			(* Case 20 - PROGRAMMA[106] ASSE Z -> TRASLAZIONE A QUOTA DI FUORI INGOMBRO *)	
			20:	
				IF StepInto THEN
					Programma_Z[Z_PosFuoriIngombroVuotoLastra].Stato 			:= DA_ESEGUIRE;
					Programma_Z[Z_PosFuoriIngombroVuotoLastra].InterpolaAsse 	:= NO_INTERPOLAZIONE_ASSE;
					ProgrammaToModule_Z 										:= Programma_Z[Z_PosFuoriIngombroVuotoLastra];
					Ciclo^.Passo := 21;
					STEPDone := FALSE;
				END_IF
				
			(* Case 21 - Attesa completamento del comando MOVETOPOS o del raggiungimento quota di Pre-Movimento se abilitata la funzione*)
			21: 
				IF Programma_Z[Z_PosFuoriIngombroVuotoLastra].Stato = TERMINATO OR
					Asse_Z_InFinestraDiPassMode OR 
					QuotaAnticipoDinamicaZ_Raggiunta THEN
					Ciclo^.Passo := 22;
					STEPDone := TRUE;
				ELSIF Programma_Z[Z_PosFuoriIngombroVuotoLastra].Stato = INTERROTTO THEN
					Ciclo^.Passo := 21;										
				END_IF
				
			(* Case 22 - Vado a quota di fuori ingombro con X *)
			22: IF Programma_Z[Z_PosFuoriIngombroVuotoLastra].Stato = INTERROTTO THEN
					Ciclo^.Passo := 22;
				ELSE
					IF StepInto THEN	
						IF FuoriIngombroXNecessario THEN
							Programma_X[X_PosFuoriIngombroVuotoLastra].Stato 			:= DA_ESEGUIRE;
							Programma_X[X_PosFuoriIngombroVuotoLastra].InterpolaAsse 	:= NO_INTERPOLAZIONE_ASSE;
							ProgrammaToModule_X 										:= Programma_X[X_PosFuoriIngombroVuotoLastra];
							Ciclo^.Passo := 23;
						ELSE
							Ciclo^.Passo := 24;
						END_IF
						STEPDone := FALSE;
					END_IF									
				END_IF

			(* Case 23 - Attendo x fuori ingombro *)
			23:
				IF Programma_Z[Z_PosFuoriIngombroVuotoLastra].Stato = INTERROTTO OR
					Programma_X[X_PosFuoriIngombroVuotoLastra].Stato = INTERROTTO THEN
						Ciclo^.Passo := 23;
				ELSIF (Programma_X[X_PosFuoriIngombroVuotoLastra].Stato = TERMINATO OR 
					Asse_X_InFinestraDiPassMode) THEN	
						Ciclo^.Passo := 24;
						STEPDone := TRUE;									
				END_IF
		
				
			(* Case 24 - Vado a quota di fuori ingombro y e j  *)
			24:
				IF Programma_Z[Z_PosFuoriIngombroVuotoLastra].Stato = INTERROTTO OR 
					Programma_X[X_PosFuoriIngombroVuotoLastra].Stato = INTERROTTO THEN
						Ciclo^.Passo := 24;										
				ELSE
					IF StepInto THEN
						Programma_Y[Y_PosFuoriIngombroVuotoLastra].Stato 			:= DA_ESEGUIRE;
						Programma_Y[Y_PosFuoriIngombroVuotoLastra].InterpolaAsse 	:= INTERPOLAZIONE_ASSE;
						ProgrammaToModule_Y 										:= Programma_Y[Y_PosFuoriIngombroVuotoLastra];

						Programma_J[J_PosStartApproccioPrelLastra].Stato 			:= DA_ESEGUIRE;
						//Programma_J[J_PosStartApproccioPrelLastra].InterpolaAsse 	:= INTERPOLAZIONE_ASSE;
						Programma_J[J_PosStartApproccioPrelLastra].InterpolaAsse 	:= No_INTERPOLAZIONE_ASSE;
						ProgrammaToModule_J 										:= Programma_J[J_PosStartApproccioPrelLastra];

						IF NOT FuoriIngombroYNecessario THEN
							Programma_X[X_PosStartLentaPrelievoLastra].Stato 			:= DA_ESEGUIRE;
							Programma_X[X_PosStartLentaPrelievoLastra].InterpolaAsse 	:= INTERPOLAZIONE_ASSE;
							ProgrammaToModule_X 										:= Programma_X[X_PosStartLentaPrelievoLastra];
							Ciclo^.Passo := 41;
						ELSE
							Ciclo^.Passo := 25;
						END_IF
						StartInterpolazioneAssi^ 	:= TRUE; //Abilito l'interpolazione degli assi
						STEPDone 					:= FALSE;
					END_IF
				END_IF
				
			(* Case 25 - *)
			25: IF Programma_Z[Z_PosFuoriIngombroVuotoLastra].Stato = INTERROTTO OR  
					(Programma_X[X_PosStartLentaPrelievoLastra].Stato = INTERROTTO and not FuoriIngombroYNecessario) OR
					Programma_Y[Y_PosFuoriIngombroVuotoLastra].Stato = INTERROTTO OR
					Programma_J[J_PosStartApproccioPrelLastra].Stato = INTERROTTO THEN
						Ciclo^.Passo := 25;
				ELSIF (Programma_Y[Y_PosFuoriIngombroVuotoLastra].Stato = TERMINATO OR 
					Asse_Y_InFinestraDiPassMode) AND 
					(Programma_J[J_PosStartApproccioPrelLastra].Stato = TERMINATO OR 
					Asse_J_InFinestraDiPassMode) THEN	
						Ciclo^.Passo := 40;
						STEPDone := TRUE;									
				END_IF
				
				
			(* Case 40 - PROGRAMMA[] ASSE  -> X TRASLAZIONE A QUOTA DI START LENTA PRELIEVO LASTRA *)	
			40:	
				IF Programma_Z[Z_PosFuoriIngombroVuotoLastra].Stato = INTERROTTO OR
					Programma_Y[Y_PosFuoriIngombroVuotoLastra].Stato = INTERROTTO OR
					Programma_J[J_PosStartApproccioPrelLastra].Stato = INTERROTTO THEN
						Ciclo^.Passo := 40;										
				ELSE
					IF StepInto THEN
						Programma_X[X_PosStartLentaPrelievoLastra].Stato 			:= DA_ESEGUIRE;
						Programma_X[X_PosStartLentaPrelievoLastra].InterpolaAsse 	:= NO_INTERPOLAZIONE_ASSE;
						ProgrammaToModule_X 										:= Programma_X[X_PosStartLentaPrelievoLastra];
												
						StartInterpolazioneAssi^ := FALSE; //Abilito l'interpolazione degli assi
						Ciclo^.Passo := 41;
						STEPDone := FALSE;
					END_IF
				END_IF
			
			(* Case 41 -   *)	
			41:	
				IF Programma_Z[Z_PosFuoriIngombroVuotoLastra].Stato = INTERROTTO OR
					Programma_Y[Y_PosFuoriIngombroVuotoLastra].Stato = INTERROTTO OR
					Programma_J[J_PosStartApproccioPrelLastra].Stato = INTERROTTO OR
					Programma_X[X_PosStartLentaPrelievoLastra].Stato = INTERROTTO THEN
						Ciclo^.Passo := 41;										
				ELSE
					STEPDone := TRUE;
					IF StepInto THEN
						Ciclo^.Passo := 42;
						STEPDone := FALSE;
					END_IF
				END_IF
				
			(* Case 42 -  Attesa completamento del comando MOVETOPOS o del raggiungimento quota di Pre-Movimento se abilitata la funzione *)
			42: 
				IF Programma_Z[Z_PosFuoriIngombroVuotoLastra].Stato = INTERROTTO OR
					Programma_Y[Y_PosFuoriIngombroVuotoLastra].Stato = INTERROTTO OR
					Programma_J[J_PosStartApproccioPrelLastra].Stato = INTERROTTO OR
					Programma_X[X_PosStartLentaPrelievoLastra].Stato = INTERROTTO THEN
						Ciclo^.Passo := 42;	
				ELSIF (Programma_X[X_PosStartLentaPrelievoLastra].Stato 	= TERMINATO OR Asse_X_InFinestraDiPassMode) AND
					(Programma_Y[Y_PosFuoriIngombroVuotoLastra].Stato		= TERMINATO OR Asse_Y_InFinestraDiPassMode) AND
					Programma_Z[Z_PosFuoriIngombroVuotoLastra].Stato 		= TERMINATO AND// OR Asse_Z_InFinestraDiPassMode AND
					(Programma_J[J_PosStartApproccioPrelLastra].Stato 		= TERMINATO OR Asse_J_InFinestraDiPassMode) THEN
						Ciclo^.Passo := 50;
						STEPDone := TRUE;							
				END_IF
							
			(* Case 50 - PROGRAMMA[101] ASSE Z -> TRASLAZIONE A QUOTA AMMESSA IN VELOCE DI PRELIEVO PACCO  *)
			50:
				IF StepInto THEN
					Programma_Z[Z_PosStartLentaPrelievoLastra].Stato 			:= DA_ESEGUIRE;
					Programma_Z[Z_PosStartLentaPrelievoLastra].InterpolaAsse 	:= NO_INTERPOLAZIONE_ASSE;
					ProgrammaToModule_Z 										:= Programma_Z[Z_PosStartLentaPrelievoLastra];
					Ciclo^.Passo := 51;
					STEPDone := FALSE;
				END_IF

			(* Case 51 -  Attesa completamento del comando MOVETOPOS o del raggiungimento quota di Pre-Movimento se abilitata la funzione *)
			51: 
				IF Programma_Z[Z_PosStartLentaPrelievoLastra].Stato = INTERROTTO OR
					Programma_Y[Y_PosFuoriIngombroVuotoLastra].Stato = INTERROTTO OR
					Programma_J[J_PosStartApproccioPrelLastra].Stato = INTERROTTO OR
					Programma_X[X_PosStartLentaPrelievoLastra].Stato = INTERROTTO THEN
						Ciclo^.Passo := 51;									
				ELSE
					IF Programma_X[X_PosStartLentaPrelievoLastra].Stato 	= TERMINATO AND
						Programma_Y[Y_PosFuoriIngombroVuotoLastra].Stato	= TERMINATO AND
						Programma_J[J_PosStartApproccioPrelLastra].Stato 	= TERMINATO AND
							(Programma_Z[Z_PosStartLentaPrelievoLastra].Stato = TERMINATO )THEN//OR Asse_Z_InFinestraDiPassMode) THEN
							Ciclo^.Passo := 90;
							STEPDone := TRUE;
					END_IF	
				END_IF
				
			52:
				IF Programma_Z[Z_PosStartLentaPrelievoLastra].Stato = INTERROTTO OR
					Programma_Y[Y_PosFuoriIngombroVuotoLastra].Stato = INTERROTTO OR
					Programma_J[J_PosStartApproccioPrelLastra].Stato = INTERROTTO OR
					Programma_X[X_PosStartLentaPrelievoLastra].Stato = INTERROTTO THEN
						Ciclo^.Passo := 52;									
				ELSE
					IF Programma_X[X_PosStartLentaPrelievoLastra].Stato 	= TERMINATO AND
						Programma_Y[Y_PosFuoriIngombroVuotoLastra].Stato	= TERMINATO AND
						Programma_J[J_PosStartApproccioPrelLastra].Stato 	= TERMINATO AND
							(Programma_Z[Z_PosStartLentaPrelievoLastra].Stato = TERMINATO )THEN
							IF StepInto THEN
								Programma_Z[Z_PosPrelievoInLentaLastra].Stato 			:= DA_ESEGUIRE;
								Programma_Z[Z_PosPrelievoInLentaLastra].InterpolaAsse 	:= NO_INTERPOLAZIONE_ASSE;
								ProgrammaToModule_Z 									:= Programma_Z[Z_PosPrelievoInLentaLastra];
								Ciclo^.Passo := 53;
								STEPDone := FALSE;
							END_IF
					END_IF	
				END_IF			
						
			53:
				IF Programma_Z[Z_PosPrelievoInLentaLastra].Stato = INTERROTTO OR
					Programma_Y[Y_PosFuoriIngombroVuotoLastra].Stato = INTERROTTO OR
					Programma_J[J_PosStartApproccioPrelLastra].Stato = INTERROTTO OR
					Programma_X[X_PosStartLentaPrelievoLastra].Stato = INTERROTTO THEN
						Ciclo^.Passo := 53;									
				ELSE
					IF Programma_X[X_PosStartLentaPrelievoLastra].Stato 	= TERMINATO AND
						Programma_Y[Y_PosFuoriIngombroVuotoLastra].Stato	= TERMINATO AND
						Programma_J[J_PosStartApproccioPrelLastra].Stato 	= TERMINATO AND
							(Programma_Z[Z_PosPrelievoInLentaLastra].Stato = TERMINATO )THEN
							Ciclo^.Passo := 90;
							STEPDone := TRUE;
					END_IF	
				END_IF

			(* Case 90 - PROGRAMMA[] ASSE Y -> TRASLAZIONE IN Y FINO ALLA QUOTA AMMESSA IN VELOCE E ATTIVAZIONE ASPIRAZIONE *)
			90:
				IF Programma_Z[Z_PosStartLentaPrelievoLastra].Stato = INTERROTTO OR
					Programma_Y[Y_PosFuoriIngombroVuotoLastra].Stato = INTERROTTO OR
					Programma_J[J_PosStartApproccioPrelLastra].Stato = INTERROTTO OR
					Programma_X[X_PosStartLentaPrelievoLastra].Stato = INTERROTTO THEN
						Ciclo^.Passo := 90; 									
				ELSE
					IF StepInto THEN
						Programma_Y[Y_PosStartLentaPrelievoLastra].Stato 			:= DA_ESEGUIRE;
						Programma_Y[Y_PosStartLentaPrelievoLastra].InterpolaAsse 	:= NO_INTERPOLAZIONE_ASSE;
						ProgrammaToModule_Y 										:= Programma_Y[Y_PosStartLentaPrelievoLastra];
						TFParametersArrayClear(ADR(ParametersArray));
						ParametersArray.Parameters[0] := BOOL_TO_STRING(NOT PrelievoPezzoOrizzontale);//SE TRUE: pezzo prelevato da cavallina, altrimenti prelievo orizzontale
						TFCommandSend(CmdPRELOAD,ParametersArray,ModulePinza^.Cmd);//LANCIO COMANDO ASPIRAZIONE PINZA
						Ciclo^.Passo := 91;
						STEPDone := FALSE;
					END_IF
				END_IF	
	
			(* Case 91 -  Attesa completamento dei comandi *)
			91: 
				IF Programma_Y[Y_PosStartLentaPrelievoLastra].Stato = INTERROTTO OR 
					TFStateCodeGet(ModulePinza^.State) = StateERROR THEN
						Ciclo^.Passo := 91; 										
				ELSE
					IF (Programma_Y[Y_PosStartLentaPrelievoLastra].Stato = TERMINATO OR Asse_Y_InFinestraDiPassMode) AND
						TFStateCodeGet(ModulePinza^.State) = StatePRELOAD_END THEN
							Ciclo^.Passo := 100;
							STEPDone := FALSE;
					END_IF	
				END_IF
				
			(* Case 100 - Lancio Tasteggio J *)
			100:
				IF StepInto THEN
					IF HMI_AbilitaTasteggioRotazionePinza THEN
						TFParametersArrayClear(ADR(ParametersArray));
						TFCommandSend(CmdTASTEGGIO,ParametersArray,ModuleAx_J^.Cmd);//LANCIO COMANDO per tateggio inclinazione pinza
					END_IF
					//!!!!!!!!!!!!!!!NB!!!!!!!!!!!	ModuleAx_J^.IN_Stop := TRUE; //Fermo Comando di tasteggio
					Ciclo^.Passo := 101;
					STEPDone := FALSE;
				END_IF

			(* Case 101 -  Attesa completamento del comando DI TASTEGGIO DELLA J*)
			101: 
				IF TFStateCodeGet(ModulePinza^.State) = StateError THEN
					Ciclo^.Passo := 101;																
				ELSE
					IF (TFStateCodeGet(ModuleAX_J^.State) >= StateTASTEGGIO_RUN + 10 AND TFStateCodeGet(ModuleAX_J^.State) <= StateTASTEGGIO_END) OR NOT HMI_AbilitaTasteggioRotazionePinza THEN		
						IF PrelievoPezzoOrizzontale THEN
							Ciclo^.Passo := 150;
						ELSE
							Ciclo^.Passo := 110;	
						END_IF

						STEPDone := TRUE;
					END_IF	
				END_IF
			
			(* Case 110 - Tasteggio in direzione Y *)
			110:
				IF Programma_Z[Z_PosStartLentaPrelievoLastra].Stato = INTERROTTO OR
					Programma_Y[Y_PosFuoriIngombroVuotoLastra].Stato = INTERROTTO OR
					Programma_J[J_PosStartApproccioPrelLastra].Stato = INTERROTTO OR
					Programma_X[X_PosStartLentaPrelievoLastra].Stato = INTERROTTO OR
					TFStateCodeGet(ModulePinza^.State) = StateError THEN
					Ciclo^.Passo := 110;																
				ELSE
					IF StepInto THEN
							
						Programma_Y[Y_PosPrelievoInLentaLastra].Stato 			:= DA_ESEGUIRE;
						Programma_Y[Y_PosPrelievoInLentaLastra].InterpolaAsse 	:= NO_INTERPOLAZIONE_ASSE;
						ProgrammaToModule_Y 									:= Programma_Y[Y_PosPrelievoInLentaLastra];
						StartInterpolazioneAssi^ := FALSE; 
						Ciclo^.Passo := 115;
						STEPDone := FALSE;
					END_IF
				END_IF	

			(* Case 115 -  Attesa completamento del comando di tasteggio IN Y *)
			115: 
				IF TFStateCodeGet(ModulePinza^.State) = StateError OR 
					Programma_Y[Y_PosPrelievoInLentaLastra].Stato = INTERROTTO	THEN
						Ciclo^.Passo := 115;																
				ELSE
					IF Programma_Y[Y_PosPrelievoInLentaLastra].Stato = TERMINATO THEN//Pezzo in presa
							Ciclo^.Passo := 116;//dichiaro il ciclo terminato
							ModuleAx_J^.IN_Stop := TRUE; //Fermo Comando di tasteggio
							STEPDone := TRUE;
					END_IF	
				END_IF

			(* Case 116 - DISTACCO LASTRA *)
			116: 
					IF StepInto THEN
						Programma_Z[Z_PosDistaccoLastraInLentaLastra].Stato 			:= DA_ESEGUIRE;
						Programma_Z[Z_PosDistaccoLastraInLentaLastra].InterpolaAsse 	:= INTERPOLAZIONE_ASSE;
						ProgrammaToModule_Z 											:= Programma_Z[Z_PosDistaccoLastraInLentaLastra];

						Programma_Y[Y_PosDistaccoLastraInLentaLastra].Stato 			:= DA_ESEGUIRE;
						Programma_Y[Y_PosDistaccoLastraInLentaLastra].InterpolaAsse 	:= INTERPOLAZIONE_ASSE;
						ProgrammaToModule_Y 											:= Programma_Y[Y_PosDistaccoLastraInLentaLastra];

						//TFParametersArrayClear(ADR(ParametersArray));
						//TFCommandSend(CmdCheckPresence,ParametersArray,ModulePinza^.Cmd);
					
						StartInterpolazioneAssi^ := TRUE; //Abilito l'interpolazione degli assi
						Ciclo^.Passo := 117;
						STEPDone := FALSE;
					END_IF	

			(* Case 117 -  Attesa completamento del comando *)
			117: 
				IF Programma_Z[Z_PosDistaccoLastraInLentaLastra].Stato = INTERROTTO OR
					Programma_Y[Y_PosDistaccoLastraInLentaLastra].Stato = INTERROTTO THEN
						Ciclo^.Passo := 117;																
				ELSE
					IF Programma_Z[Z_PosDistaccoLastraInLentaLastra].Stato = TERMINATO AND 
						Programma_Y[Y_PosDistaccoLastraInLentaLastra].Stato = TERMINATO THEN //AND 
						//TFStateCodeGet(ModulePinza^.State) = StateCHECKPRESENCE_END THEN
						TFParametersArrayClear(ADR(ParametersArray));
						TFCommandSend(CmdCheckPresence,ParametersArray,ModulePinza^.Cmd);
						Ciclo^.Passo := 118;//1000;//CICLO TERMINATO
					END_IF
				END_IF

			(* Case 118 -  Attesa completamento del comando *)
			118:
				IF TFStateCodeGet(ModulePinza^.State) = StateCHECKPRESENCE_END THEN
					IF	ModulePinza^.StatoPinza.ElementoPrelevato THEN
						IF StepInto THEN
							Ciclo^.Passo := 1000;//CICLO TERMINATO
							ModuleAx_J^.IN_Stop := TRUE; //Fermo Comando di tasteggio
							STEPDone := FALSE;
							SupportoVuoto := FALSE;
						END_IF
					ELSIF NOT ModulePinza^.StatoPinza.ElementoPrelevato THEN
						IF NumeroTentativiPresaAttuali >= NumeroTentativiPresa THEN
							SupportoVuoto := TRUE;
							IF StepInto THEN
								Ciclo^.Passo := 1000;//CICLO TERMINATO
								ModuleAx_J^.IN_Stop := TRUE; //Fermo Comando di tasteggio
								STEPDone := FALSE;
							END_IF
						ELSE
							SupportoVuoto := FALSE;
							Ciclo^.Passo := 50;//torno a fare prelievo     52??
							NumeroTentativiPresaAttuali := NumeroTentativiPresaAttuali+1;
						END_IF
					END_IF
				ELSIF TFStateCodeGet(ModulePinza^.State) = StateERROR THEN
					Ciclo^.Passo := 118;
				END_IF	
				
			(* Case 150 - Tasteggio in direzione Z *)
			150: 
				IF Programma_Z[Z_PosStartLentaPrelievoLastra].Stato = INTERROTTO OR
					Programma_Y[Y_PosPrelievoInLentaLastra].Stato = INTERROTTO OR
					Programma_J[J_PosStartApproccioPrelLastra].Stato = INTERROTTO OR
					Programma_X[X_PosStartLentaPrelievoLastra].Stato = INTERROTTO THEN
						Ciclo^.Passo := 150;									
				ELSE
					
					IF StepInto THEN
						Programma_Z[Z_PosPrelievoInLentaLastra].Stato 			:= DA_ESEGUIRE;
						Programma_Z[Z_PosPrelievoInLentaLastra].InterpolaAsse 	:= NO_INTERPOLAZIONE_ASSE;
						ProgrammaToModule_Z 									:= Programma_Z[Z_PosPrelievoInLentaLastra];
	
						Ciclo^.Passo := 155;
						STEPDone := FALSE;
					END_IF	
				END_IF
		
			(* Case 155 -  Attesa completamento del comando del tasteggio IN Z *)
			155: 
				IF TFStateCodeGet(ModulePinza^.State) = StateError OR 
					Programma_Z[Z_PosPrelievoInLentaLastra].Stato = INTERROTTO	THEN
						Ciclo^.Passo := 155;																
				ELSE
					IF Programma_Z[Z_PosPrelievoInLentaLastra].Stato = TERMINATO THEN//Pezzo in presa
						Ciclo^.Passo := 156;//VADO A ESEGUIRE IL DISTACCO LASTRA
						ModuleAx_J^.IN_Stop := TRUE; //Fermo Comando di tasteggio
						//TFParametersArrayClear(ADR(ParametersArray));
						//TFCommandSend(CmdCheckPresence,ParametersArray,ModulePinza^.Cmd);
						IF NumeroTentativiPresaAttuali = 0 THEN
							Programma_Z[Z_PosDistaccoLastraInLentaLastra].Quota_Destinazione := ModuleAX_Z^.QuotaAsseLetturaTasteggio + OffsetDistacco.Lastra.Z;
						ELSE
							Programma_Z[Z_PosDistaccoLastraInLentaLastra].Quota_Destinazione := ModuleAX_Z^.QuotaAsseLetturaTasteggio + OffsetDistacco.Lastra.Z+100;
						END_IF
						//
						
						RichiestaEspulsionePerPolistirolo := FALSE;
						IF ModuleAX_Z^.QuotaAsseLetturaTasteggio <= (WorkArea[Mission.PPick].Z + 1100) THEN
							idxTasteg := idxTasteg+1;
							IF idxTasteg > 10 THEN
								idxTasteg := 1;
								MemoriaQuoteTasteggio := MemoriaQuoteTasteggioVuoto;
							END_IF
							MemoriaQuoteTasteggio[idxTasteg] := ModuleAX_Z^.QuotaAsseLetturaTasteggio;
							IF (idxTasteg >= HMI_NumeroTentativiPolistiroloSuPallet)THEN
								FOR i := 1 TO HMI_NumeroTentativiPolistiroloSuPallet DO
									IF ModuleAX_Z^.QuotaAsseLetturaTasteggio <= MemoriaQuoteTasteggio[i]+2 THEN
										RichiestaEspulsionePerPolistirolo := TRUE;
										//Errore := ErrMalfunzionamentoSensoriPresenzaPinza;
										idxTasteg := 0;
										MemoriaQuoteTasteggio := MemoriaQuoteTasteggioVuoto;
									END_IF
								END_FOR
							END_IF
						ELSE
							idxTasteg := 0;
							MemoriaQuoteTasteggio := MemoriaQuoteTasteggioVuoto;
						END_IF
						
						STEPDone := TRUE;
					END_IF	
				END_IF

			(* Case 156 - Sfogliatura J *)
			156: 
					IF StepInto THEN
						Programma_Z[Z_PosDistaccoLastraInLentaLastra].Stato 			:= DA_ESEGUIRE;
						Programma_Z[Z_PosDistaccoLastraInLentaLastra].InterpolaAsse 	:= NO_INTERPOLAZIONE_ASSE;
						ProgrammaToModule_Z 											:= Programma_Z[Z_PosDistaccoLastraInLentaLastra];
						IF HMI_AbilitaSfogliaturaJ THEN
							Programma_J[J_PosSfogliatura].Stato 			:= DA_ESEGUIRE;
							Programma_J[J_PosSfogliatura].InterpolaAsse 	:= NO_INTERPOLAZIONE_ASSE;
							ProgrammaToModule_J 							:= Programma_J[J_PosSfogliatura];
						END_IF			
						TFTimerSet(ADR(TimerAttesaCadutaLastra),HMI_TempoAttesaPartenzaDopoPrelievo, TRUE);			
						Ciclo^.Passo := 157;
						STEPDone := FALSE;
					END_IF	
					
			157:
				IF Programma_Z[Z_PosDistaccoLastraInLentaLastra].Stato = INTERROTTO OR Programma_Z[J_PosSfogliatura].Stato = INTERROTTO	THEN
					Ciclo^.Passo := 157;																
				ELSE	
					IF Programma_Z[Z_PosDistaccoLastraInLentaLastra].Stato = TERMINATO AND TFTimerDone(ADR(TimerAttesaCadutaLastra)) THEN
						TFParametersArrayClear(ADR(ParametersArray));
						TFCommandSend(CmdCheckPresence,ParametersArray,ModulePinza^.Cmd);
						Ciclo^.Passo := 158;	
					END_IF
				END_IF	
					

			(* Case 158 -  Attesa completamento del comando *)
			158: 
				IF Programma_Z[Z_PosDistaccoLastraInLentaLastra].Stato = INTERROTTO OR Programma_Z[J_PosSfogliatura].Stato = INTERROTTO	THEN
						Ciclo^.Passo := 158;																
				ELSE
					//TFTimerSet(ADR(TimerAttesaCadutaLastra),HMI_TempoAttesaPartenzaDopoPrelievo, (Programma_Z[Z_PosDistaccoLastraInLentaLastra].Stato <> TERMINATO));
					IF Programma_Z[Z_PosDistaccoLastraInLentaLastra].Stato = TERMINATO AND TFTimerDone(ADR(TimerAttesaCadutaLastra)) AND
						TFStateCodeGet(ModulePinza^.State) = StateCHECKPRESENCE_END AND (Programma_J[J_PosSfogliatura].Stato = TERMINATO OR NOT HMI_AbilitaSfogliaturaJ) THEN
						IF ModulePinza^.StatoPinza.ElementoPrelevato AND NOT RichiestaEspulsionePerPolistirolo THEN
							Ciclo^.Passo := 1000;//CICLO TERMINATO
								
							ModuleAx_J^.IN_Stop := TRUE; //Fermo Comando di tasteggio
							STEPDone := FALSE;
							SupportoVuoto := FALSE;
							IF //((ModulePinza^.StatoPinza.LatoSxPiastrellaInPresa or ModulePinza^.StatoPinza.LatoDxPiastrellaInPresa) //AND 
								//(ModulePinza^.StatoPinza.LatoDxFaldaInPresa OR ModulePinza^.StatoPinza.LatoSxFaldaInPresa)) OR 
								(ModulePinza^.StatoPinza.LatoSxPiastrellaInPresa AND WorkAreaState[Mission.PPick].TransportState.Supporto.Tipologia = PALLET_STANDARD AND WorkAreaState[Mission.PPick].TransportState.Supporto.XDim < 1400 )OR
								(ModulePinza^.StatoPinza.LatoSxPiastrellaInPresa AND ModulePinza^.StatoPinza.LatoDxPiastrellaInPresa) THEN
									idxTasteg := 0;
									MemoriaQuoteTasteggio := MemoriaQuoteTasteggioVuoto;
							END_IF		
						ELSIF NOT ModulePinza^.StatoPinza.ElementoPrelevato OR (RichiestaEspulsionePerPolistirolo AND ModuleAX_Z^.QuotaAsseLetturaTasteggio <= (WorkArea[Mission.PPick].Z + HMI_AltezzaControlloPolistirolo)) THEN
							IF NumeroTentativiPresaAttuali >= NumeroTentativiPresa OR RichiestaEspulsionePerPolistirolo THEN
								idxTasteg := 0;
								MemoriaQuoteTasteggio := MemoriaQuoteTasteggioVuoto;
								SupportoVuoto := TRUE;
								RichiestaEspulsionePerPolistirolo := FALSE;
								IF StepInto THEN
									Ciclo^.Passo := 1000;//CICLO TERMINATO
									ModuleAx_J^.IN_Stop := TRUE; //Fermo Comando di tasteggio
									STEPDone := FALSE;
								END_IF
							ELSE
								SupportoVuoto := FALSE;
								Ciclo^.Passo := 150;//torno a fare prelievo
								NumeroTentativiPresaAttuali := NumeroTentativiPresaAttuali+1;
							END_IF
						ELSIF RichiestaEspulsionePerPolistirolo THEN
							idxTasteg := 0;
							MemoriaQuoteTasteggio := MemoriaQuoteTasteggioVuoto;
							RichiestaEspulsionePerPolistirolo := FALSE;
							Errore := ErrMalfunzionamentoSensoriPresenzaPinza;
						END_IF	
					END_IF
				END_IF	

			(* Case 159 - SFOGLIO J *)
			159: 
				IF StepInto THEN
					
					Programma_J[J_PosSfogliatura].Stato 			:= DA_ESEGUIRE;
					Programma_J[J_PosSfogliatura].InterpolaAsse 	:= NO_INTERPOLAZIONE_ASSE;
					ProgrammaToModule_J 							:= Programma_J[J_PosSfogliatura];
	
					Ciclo^.Passo := 159;
					STEPDone := FALSE;
				END_IF	

			(* Case 160 - FINE SFOGLIO J *)
			160:
				IF Programma_Z[J_PosSfogliatura].Stato = INTERROTTO	THEN
						Ciclo^.Passo := 160;																
				ELSE
					IF Programma_Z[J_PosSfogliatura].Stato = TERMINATO THEN//Pezzo in presa
						Ciclo^.Passo 		:= 1000;//termino ciclo
						ModuleAx_J^.IN_Stop := TRUE; //Fermo Comando di tasteggio
						STEPDone := TRUE;
					END_IF	
				END_IF

			(* Case 1000 *)
			1000:
				STEPDone := TRUE;
				Ciclo^.Stato := TERMINATO;
				Ciclo^.Passo := 1000;
				
			(* Case 9999 - Ciclo NON annullato o NON terminato*)
			9999:
				Ciclo^.Stato := INTERROTTO;
				Ciclo^.Passo := 9999;
	ELSE						
		;	
	END_CASE;
ELSE								//Se il ciclo deve essere interrotto, setto il suo nuovo stato
	Ciclo^.Stato := INTERROTTO;
END_IF

END_FUNCTION_BLOCK

// ---- POUs/TFCicliDiLavoro/Lastre/Cicli Depallettizzatore/TFCiclo_Deposito_Lastra_Depal.TcPOU
FUNCTION_BLOCK TFCiclo_Deposito_Lastra_Depal
VAR_INPUT
	Ciclo 		: POINTER TO Stato_Ciclo_Lavoro;
	Programma : POINTER TO TFProgramma_Ciclo_Lastra;
	ModuleAX_X : POINTER TO TFModulePalletizer_Ax;
	ModuleAX_Y : POINTER TO TFModulePalletizer_Ax;
	ModuleAX_Z : POINTER TO TFModulePalletizer_Ax;
	ModuleAX_J : POINTER TO TFModulePalletizer_AxJ_Lastre;
	ModulePinza : POINTER TO TFModulePalletizer_Pinza;
	StartInterpolazioneAssi : POINTER TO BOOL;
	QuotaPassModePuntoIntermedio : ARRAY [1..3] OF REAL;
	AbilitazioneGlobalePassMode	: BOOL;
	InterrompiCiclo : BOOL;
	Abilita_Ciclo_Step : BOOL;
	Command_Step : BOOL;
	AbilitazioneAnticipoDinamicoMovimenti : BOOL;
	
END_VAR
VAR_OUTPUT
	STEPDone	: BOOL;
	//MaterialeDepositatoSuLinea : BOOL;
END_VAR
VAR
	ConAccostamentoZ : BOOL := FALSE;
	StepInto: BOOL;
END_VAR

(* Set della variabile che mi permette di fare lo STEP nel ciclo *)
StepInto := (Abilita_Ciclo_Step AND Command_Step) OR NOT Abilita_Ciclo_Step;

(* Reset Anticipo Dinamico se non ho l'abilitazione *)
IF NOT AbilitazioneAnticipoDinamicoMovimenti OR NOT HMI_DisabilitaAnticipiGLOBALE THEN
	QuotaAnticipoDinamicaX_Raggiunta := FALSE;
	QuotaAnticipoDinamicaY_Raggiunta := FALSE;
	QuotaAnticipoDinamicaZ_Raggiunta := FALSE;
END_IF

IF NOT InterrompiCiclo THEN
	IF Ciclo^.Stato = TERMINATO OR Ciclo^.Stato = ANNULLATO THEN
		Ciclo^.Passo := 0;
	ELSIF Ciclo^.Stato = INTERROTTO AND Ciclo^.Passo = 56 THEN
		Ciclo^.Passo := 56;
	ELSIF Ciclo^.Stato = INTERROTTO AND NOT Ciclo^.Passo = 56 THEN
		Ciclo^.Passo := 999;
	END_IF
	Ciclo^.Stato := IN_ESECUZIONE;
	CASE Ciclo^.Passo OF
			(* Case 0 *)
			0:  Ciclo^.Stato := IN_ESECUZIONE;
				Ciclo^.Passo := 10;
				STEPDone := FALSE;
				
			(* Case 10 -  *)
			10:	MaterialeDepositatoSuLinea := FALSE;
				Ciclo^.Passo := 20;
				
						
			(* Case 20 - PROGRAMMA[Z_PosFuoriIngombroCaricoLastra] ASSE Z -> TRASLAZIONE A QUOTA DI FUORI INGOMBRO CON lLASTRA A BORDO *)	
			20:	Ciclo^.Stato := IN_ESECUZIONE;
				IF StepInto THEN
					Programma_Z[Z_PosFuoriIngombroCaricoLastra].Stato 			:= DA_ESEGUIRE;
					Programma_Z[Z_PosFuoriIngombroCaricoLastra].InterpolaAsse 	:= NO_INTERPOLAZIONE_ASSE;
					ProgrammaToModule_Z 										:= Programma_Z[Z_PosFuoriIngombroCaricoLastra];
					Ciclo^.Passo := 21;
					STEPDone := FALSE;
				END_IF
				
			(* Case 21 - Attesa completamento del comando MOVETOPOS o del raggiungimento quota di Pre-Movimento se abilitata la funzione*)
			21: 
				IF Programma_Z[Z_PosFuoriIngombroCaricoLastra].Stato = INTERROTTO THEN
					Ciclo^.Passo := 21;		
				ELSIF Programma_Z[Z_PosFuoriIngombroCaricoLastra].Stato = TERMINATO OR
					Asse_Z_InFinestraDiPassMode THEN
					Ciclo^.Passo := 22; //Eseguo prima il Fuori Ingombro colonne con la J poi il resto dei posizionamenti
					STEPDone := TRUE;							
				END_IF
				
			22: IF Programma_Z[Z_PosFuoriIngombroCaricoLastra].Stato = INTERROTTO THEN
					 Ciclo^.Passo := 22;
				ELSIF Programma_Z[Z_PosFuoriIngombroCaricoLastra].Stato = TERMINATO OR 
						Asse_Z_InFinestraDiPassMode OR 
						QuotaAnticipoDinamicaZ_Raggiunta THEN
							IF StepInto THEN
								Programma_J[J_PosFuoriIngombro].Stato 			:= DA_ESEGUIRE;
								Programma_J[J_PosFuoriIngombro].InterpolaAsse 	:= NO_INTERPOLAZIONE_ASSE;
								ProgrammaToModule_J		 						:= Programma_J[J_PosFuoriIngombro];
								Ciclo^.Passo := 23;
								STEPDone := FALSE;
							END_IF									
				END_IF
			
			23: IF Programma_Z[Z_PosFuoriIngombroCaricoLastra].Stato = INTERROTTO OR 
					Programma_J[J_PosFuoriIngombro].Stato = INTERROTTO THEN
					 Ciclo^.Passo := 23;
				ELSIF (Programma_Z[Z_PosFuoriIngombroCaricoLastra].Stato = TERMINATO OR Asse_Z_InFinestraDiPassMode (*OR QuotaAnticipoDinamicaZ_Raggiunta*)) AND 
					(Programma_J[J_PosFuoriIngombro].Stato = TERMINATO OR Asse_J_InFinestraDiPassMode OR QuotaAnticipoDinamicaJ_Raggiunta) THEN
						Ciclo^.Passo := 24;
						STEPDone := TRUE;										
				END_IF	
							
				
			(* Case 24 - Scelgo in quale direzione devo muovermi per primo a seconda della disposizione delle postazioni *)	
			24:	
				CASE ASSE_DISPOSIZIONE_POSTAZIONI OF
					
					LUNGO_X:
							Ciclo^.Passo := 25;
				
					LUNGO_Y:	
							IF FuoriIngombroXNecessario THEN
								IF FuoriIngombroYNecessario THEN
									Ciclo^.Passo := 25;
								ELSE
									Ciclo^.Passo := 50;
								END_IF
								
							ELSE
								Ciclo^.Passo := 52;
							END_IF
			
				END_CASE
				
			(* Case 25 - Vado a quota di fuori ingombro con Y *)
			25:	IF Programma_Z[Z_PosFuoriIngombroCaricoLastra].Stato = INTERROTTO OR
					Programma_J[J_PosFuoriIngombro].Stato = INTERROTTO THEN
						Ciclo^.Passo := 25;										
				ELSE
					IF StepInto THEN
						Programma_Y[Y_PosFuoriIngombroCaricoLastra].Stato 			:= DA_ESEGUIRE;
						Programma_Y[Y_PosFuoriIngombroCaricoLastra].InterpolaAsse 	:= NO_INTERPOLAZIONE_ASSE;
						ProgrammaToModule_Y 										:= Programma_Y[Y_PosFuoriIngombroCaricoLastra];
						Ciclo^.Passo := 26;
						STEPDone := FALSE;
					END_IF
				END_IF
					
			(* Case 26 - Check se a quota di fuori ingombro con Y *)		
			26:	IF Programma_Y[Y_PosFuoriIngombroCaricoLastra].Stato = INTERROTTO OR 
					Programma_Z[Z_PosFuoriIngombroCaricoLastra].Stato = INTERROTTO OR 
					Programma_J[J_PosFuoriIngombro].Stato = INTERROTTO THEN
						Ciclo^.Passo := 26;
				ELSE	
					IF Programma_Y[Y_PosFuoriIngombroCaricoLastra].Stato = TERMINATO OR 
						Asse_Y_InFinestraDiPassMode THEN
							Ciclo^.Passo := 30;
							STEPDone := TRUE;							
					END_IF
				END_IF
										
			(* Case 30 - PROGRAMMA[0] ASSE X  -> TRASLAZIONE A QUOTA DI DEPOSITO  *)	
			30:	IF Programma_Z[Z_PosFuoriIngombroCaricoLastra].Stato = INTERROTTO OR 
					Programma_Y[Y_PosFuoriIngombroCaricoLastra].Stato = INTERROTTO OR 
					Programma_J[J_PosFuoriIngombro].Stato = INTERROTTO THEN
						Ciclo^.Passo := 30;										
				ELSE
					IF StepInto THEN
						Programma_X[X_PosStartLentaDepositoLastra].Stato 			:= DA_ESEGUIRE;
						Programma_X[X_PosStartLentaDepositoLastra].InterpolaAsse 	:= NO_INTERPOLAZIONE_ASSE;
						ProgrammaToModule_X 										:= Programma_X[X_PosStartLentaDepositoLastra];
					
						Ciclo^.Passo := 31;
						STEPDone := FALSE;
					END_IF
				END_IF			
				
			(* Case 31 -  Attesa completamento del comando MOVETOPOS o del raggiungimento quota di Pre-Movimento se abilitata la funzione *)
			31: 
				IF Programma_X[X_PosStartLentaDepositoLastra].Stato = INTERROTTO OR
					Programma_Y[Y_PosFuoriIngombroCaricoLastra].Stato = INTERROTTO OR
					Programma_Z[Z_PosFuoriIngombroCaricoLastra].Stato = INTERROTTO OR 
					Programma_J[J_PosFuoriIngombro].Stato = INTERROTTO THEN
						Ciclo^.Passo := 31;
				ELSE	
					IF (Programma_X[X_PosStartLentaDepositoLastra].Stato = TERMINATO OR Asse_X_InFinestraDiPassMode OR QuotaAnticipoDinamicaX_Raggiunta) THEN 
						Ciclo^.Passo := 32;
						STEPDone := TRUE;							
					END_IF
				END_IF
				
			(* Case 32 - Vado a quota di START LENTA CON GLI ASSI con Y,Z,J *)
			32:
				IF Programma_X[X_PosStartLentaDepositoLastra].Stato = INTERROTTO OR
					Programma_Y[Y_PosFuoriIngombroCaricoLastra].Stato = INTERROTTO OR
					Programma_Z[Z_PosFuoriIngombroCaricoLastra].Stato = INTERROTTO OR 
					Programma_J[J_PosFuoriIngombro].Stato = INTERROTTO THEN
						Ciclo^.Passo := 32;										
				ELSE
					IF StepInto THEN
						TFParametersArrayClear(ADR(ParametersArray));
						Programma_Y[Y_PosStartLentaDepositoLastra].Stato 			:= DA_ESEGUIRE;
						Programma_Y[Y_PosStartLentaDepositoLastra].InterpolaAsse 	:= INTERPOLAZIONE_ASSE;
						ProgrammaToModule_Y 										:= Programma_Y[Y_PosStartLentaDepositoLastra];
				
						Programma_Z[Z_PosStartLentaDepositoLastra].Stato 			:= DA_ESEGUIRE;
						Programma_Z[Z_PosStartLentaDepositoLastra].InterpolaAsse 	:= INTERPOLAZIONE_ASSE;
						ProgrammaToModule_Z 										:= Programma_Z[Z_PosStartLentaDepositoLastra];
						
						Programma_J[J_PosDepositoLastra].Stato 						:= DA_ESEGUIRE;
						Programma_J[J_PosDepositoLastra].InterpolaAsse 				:= INTERPOLAZIONE_ASSE;
						ProgrammaToModule_J 										:= Programma_J[J_PosDepositoLastra];
						
						StartInterpolazioneAssi^ := TRUE; //Abilito l'interpolazione degli assi
												
						Ciclo^.Passo := 33;
						STEPDone := FALSE;
					END_IF
				END_IF
			
			(* Case 33 - Attendo completamento comando o assi in finsetra *)
			33:
				IF Programma_Y[Y_PosStartLentaDepositoLastra].Stato = TERMINATO (*OR Asse_Y_InFinestraDiPassMode)*) AND 
					Programma_J[J_PosDepositoLastra].Stato = TERMINATO (*OR Asse_J_InFinestraDiPassMode)*) AND
					Programma_X[X_PosStartLentaDepositoLastra].Stato = TERMINATO (*OR Asse_X_InFinestraDiPassMode)*) AND 
					Programma_Z[Z_PosStartLentaDepositoLastra].Stato = TERMINATO (*OR Asse_Z_InFinestraDiPassMode)*) THEN
						Ciclo^.Passo := 34;
						STEPDone := TRUE;
				ELSIF Programma_Y[Y_PosStartLentaDepositoLastra].Stato = INTERROTTO OR 
					Programma_J[J_PosDepositoLastra].Stato = INTERROTTO OR 
					Programma_X[X_PosStartLentaDepositoLastra].Stato = INTERROTTO OR
					Programma_Z[Z_PosStartLentaDepositoLastra].Stato = TERMINATO THEN

						Ciclo^.Passo := 33;								
				END_IF

			(* Case 34 - Vado a quota di finale con Z *)
			34:
				IF Programma_X[X_PosStartLentaDepositoLastra].Stato = INTERROTTO OR
					Programma_Y[Y_PosFuoriIngombroCaricoLastra].Stato = INTERROTTO OR
					Programma_Z[Z_PosFuoriIngombroCaricoLastra].Stato = INTERROTTO OR 
					Programma_J[J_PosFuoriIngombro].Stato = INTERROTTO THEN
						Ciclo^.Passo := 34;										
				ELSE
					IF StepInto THEN
						TFParametersArrayClear(ADR(ParametersArray));
						//Programma_Y[Y_PosDepositoInLentaLastra].Stato 			:= DA_ESEGUIRE;
						//Programma_Y[Y_PosDepositoInLentaLastra].InterpolaAsse 	:= INTERPOLAZIONE_ASSE;
						//ProgrammaToModule_Y 									:= Programma_Y[Y_PosDepositoInLentaLastra];
				
						Programma_Z[Z_PosDepositoInLentaLastra].Stato 			:= DA_ESEGUIRE;
						Programma_Z[Z_PosDepositoInLentaLastra].InterpolaAsse 	:= INTERPOLAZIONE_ASSE;
						ProgrammaToModule_Z 									:= Programma_Z[Z_PosDepositoInLentaLastra];
												
						StartInterpolazioneAssi^ := TRUE; //Abilito l'interpolazione degli assi
												
						Ciclo^.Passo := 35;
						STEPDone := FALSE;
					END_IF
				END_IF

			(* Case 35 - Attendo completamento comando o assi in finsetra *)
			35:
				IF //Programma_Y[Y_PosStartLentaDepositoLastra].Stato = TERMINATO (*OR Asse_Y_InFinestraDiPassMode)*) AND 
					//Programma_J[J_PosDepositoLastra].Stato = TERMINATO (*OR Asse_J_InFinestraDiPassMode)*) AND
					//Programma_X[X_PosStartLentaDepositoLastra].Stato = TERMINATO (*OR Asse_X_InFinestraDiPassMode)*) AND 
					Programma_Z[Z_PosDepositoInLentaLastra].Stato = TERMINATO (*OR Asse_Z_InFinestraDiPassMode)*) THEN
						Ciclo^.Passo := 90;
						STEPDone := TRUE;
				ELSIF //Programma_Y[Y_PosStartLentaDepositoLastra].Stato = INTERROTTO OR 
					//Programma_J[J_PosDepositoLastra].Stato = INTERROTTO OR 
					//Programma_X[X_PosStartLentaDepositoLastra].Stato = INTERROTTO OR
					Programma_Z[Z_PosDepositoInLentaLastra].Stato = INTERROTTO THEN
						Ciclo^.Passo := 35;								
				END_IF
										
			(* Case 50 - Vado a quota di deposito con X *)
			50:	IF Programma_Z[Z_PosFuoriIngombroCaricoLastra].Stato = INTERROTTO OR
					Programma_J[J_PosFuoriIngombro].Stato = INTERROTTO THEN
						Ciclo^.Passo := 50;										
				ELSE
					IF StepInto THEN
						Programma_X[X_PosStartLentaDepositoLastra].Stato 			:= DA_ESEGUIRE;
						Programma_X[X_PosStartLentaDepositoLastra].InterpolaAsse 	:= NO_INTERPOLAZIONE_ASSE;
						ProgrammaToModule_X 										:= Programma_X[X_PosStartLentaDepositoLastra];
						Ciclo^.Passo := 51;
						STEPDone := FALSE;
					END_IF
				END_IF
					
			(* Case 51 - Check se a quota di deposito X *)		
			51:	IF Programma_X[X_PosStartLentaDepositoLastra].Stato = INTERROTTO OR 
					Programma_Z[Z_PosFuoriIngombroCaricoLastra].Stato = INTERROTTO OR 
					Programma_J[J_PosFuoriIngombro].Stato = INTERROTTO THEN
						Ciclo^.Passo := 51;
				ELSE	
					IF Programma_X[X_PosStartLentaDepositoLastra].Stato = TERMINATO OR 
						Asse_X_InFinestraDiPassMode THEN
							Ciclo^.Passo := 52;
							STEPDone := TRUE;							
					END_IF
				END_IF
										
			(* Case 52 - lancio posizionamento Y,j e x se non serve fuori ingombro  *)	
			52:	IF Programma_Z[Z_PosFuoriIngombroCaricoLastra].Stato = INTERROTTO OR 
					(Programma_X[X_PosStartLentaDepositoLastra].Stato = INTERROTTO AND FuoriIngombroXNecessario) OR 
					Programma_J[J_PosFuoriIngombro].Stato = INTERROTTO THEN
						Ciclo^.Passo := 52;										
				ELSE
					IF StepInto THEN
			
						IF NOT FuoriIngombroXNecessario THEN
							Programma_X[X_PosStartLentaDepositoLastra].Stato 			:= DA_ESEGUIRE;
							Programma_X[X_PosStartLentaDepositoLastra].InterpolaAsse 	:= INTERPOLAZIONE_ASSE;
							ProgrammaToModule_X 										:= Programma_X[X_PosStartLentaDepositoLastra];
						END_IF
					
						Programma_Y[Y_PosStartLentaDepositoLastra].Stato 			:= DA_ESEGUIRE;
						Programma_Y[Y_PosStartLentaDepositoLastra].InterpolaAsse 	:= INTERPOLAZIONE_ASSE;
						ProgrammaToModule_Y 										:= Programma_Y[Y_PosStartLentaDepositoLastra];
						
						//Programma_Z[Z_PosStartLentaDepositoLastra].Stato 			:= DA_ESEGUIRE;
						//Programma_Z[Z_PosStartLentaDepositoLastra].InterpolaAsse 	:= INTERPOLAZIONE_ASSE;
						//ProgrammaToModule_Z 										:= Programma_Z[Z_PosStartLentaDepositoLastra];
					
					
						Programma_J[J_PosDepositoLastra].Stato 						:= DA_ESEGUIRE;
						Programma_J[J_PosDepositoLastra].InterpolaAsse 				:= INTERPOLAZIONE_ASSE;
						ProgrammaToModule_J 										:= Programma_J[J_PosDepositoLastra];
			
						StartInterpolazioneAssi^ := TRUE; //Abilito l'interpolazione degli assi

						Ciclo^.Passo := 53;
						STEPDone := FALSE;
					END_IF
				END_IF			
				
			(* Case 53 -  Attesa completamento del comando MOVETOPOS o del raggiungimento quota di Pre-Movimento se abilitata la funzione *)
			53: 
				IF Programma_X[X_PosStartLentaDepositoLastra].Stato = INTERROTTO OR
					Programma_Y[Y_PosStartLentaDepositoLastra].Stato = INTERROTTO OR
					Programma_Z[Z_PosFuoriIngombroCaricoLastra].Stato = INTERROTTO OR 
					Programma_J[J_PosDepositoLastra].Stato = INTERROTTO THEN
						Ciclo^.Passo := 53;
				ELSE	
					IF (Programma_Y[Y_PosStartLentaDepositoLastra].Stato = TERMINATO OR Asse_Y_InFinestraDiPassMode OR QuotaAnticipoDinamicaY_Raggiunta) AND
						(Programma_J[J_PosDepositoLastra].Stato = TERMINATO OR Asse_J_InFinestraDiPassMode OR QuotaAnticipoDinamicaJ_Raggiunta)  THEN 
							
							Ciclo^.Passo := 54;
							STEPDone := TRUE;							
					END_IF
				END_IF
				
			(* Case 54 - Vado a quota di START LENTA CON GLI ASSI Z*)
			54:
				IF Programma_X[X_PosStartLentaDepositoLastra].Stato = INTERROTTO OR
					Programma_Y[Y_PosStartLentaDepositoLastra].Stato = INTERROTTO OR
					//Programma_Z[Z_PosStartLentaDepositoLastra].Stato = INTERROTTO OR 
					Programma_J[J_PosDepositoLastra].Stato = INTERROTTO THEN
						Ciclo^.Passo := 54;										
				ELSE
					IF StepInto THEN
						Programma_Z[Z_PosStartLentaDepositoLastra].Stato 			:= DA_ESEGUIRE;
						Programma_Z[Z_PosStartLentaDepositoLastra].InterpolaAsse 	:= NO_INTERPOLAZIONE_ASSE;
						ProgrammaToModule_Z 										:= Programma_Z[Z_PosStartLentaDepositoLastra];
								
						Ciclo^.Passo := 55;
						STEPDone := FALSE;
					END_IF
				END_IF
			
			(* Case 55 - Attendo completamento comando o assi in finsetra *)
			55:
				IF Programma_Y[Y_PosStartLentaDepositoLastra].Stato = TERMINATO (*OR Asse_Y_InFinestraDiPassMode)*) AND 
					Programma_J[J_PosDepositoLastra].Stato = TERMINATO (*OR Asse_J_InFinestraDiPassMode)*) AND
					Programma_X[X_PosStartLentaDepositoLastra].Stato = TERMINATO (*OR Asse_X_InFinestraDiPassMode)*) AND 
					Programma_Z[Z_PosStartLentaDepositoLastra].Stato = TERMINATO OR Asse_Z_InFinestraDiPassMode THEN
						Ciclo^.Passo := 56;
						StopDepositoPerArresto := TRUE;
						STEPDone := TRUE;
				ELSIF Programma_X[X_PosStartLentaDepositoLastra].Stato = INTERROTTO OR
					Programma_Y[Y_PosStartLentaDepositoLastra].Stato = INTERROTTO OR
					Programma_Z[Z_PosFuoriIngombroCaricoLastra].Stato = INTERROTTO OR 
					Programma_J[J_PosDepositoLastra].Stato = INTERROTTO THEN
						Ciclo^.Passo := 55;
				END_IF

			(* Case 56 - Vado a quota di finale con Y,Z,J *)
			56:
				IF Programma_X[X_PosStartLentaDepositoLastra].Stato = INTERROTTO OR
					Programma_Y[Y_PosFuoriIngombroCaricoLastra].Stato = INTERROTTO OR
					Programma_Z[Z_PosFuoriIngombroCaricoLastra].Stato = INTERROTTO OR 
					Programma_J[J_PosFuoriIngombro].Stato = INTERROTTO THEN
						Ciclo^.Passo := 56;										
				ELSE
					IF StepInto THEN
						TFParametersArrayClear(ADR(ParametersArray));
						RichiestaDepositoALinea := TRUE;
						StopDepositoPerArresto := TRUE;
						IF OkDepositoDaLinea THEN
							Programma_Z[Z_PosDepositoInLentaLastra].Stato 			:= DA_ESEGUIRE;
							Programma_Z[Z_PosDepositoInLentaLastra].InterpolaAsse 	:= NO_INTERPOLAZIONE_ASSE;
							ProgrammaToModule_Z 									:= Programma_Z[Z_PosDepositoInLentaLastra];						
							Ciclo^.Passo := 57;
							STEPDone := FALSE;
						END_IF						
						//StartInterpolazioneAssi^ := TRUE; //Abilito l'interpolazione degli assi
						
					END_IF
				END_IF

			(* Case 57 - Attendo completamento comando o assi in finsetra *)
			57:
				IF //Programma_Y[Y_PosStartLentaDepositoLastra].Stato = TERMINATO (*OR Asse_Y_InFinestraDiPassMode)*) AND 
					//Programma_J[J_PosDepositoLastra].Stato = TERMINATO (*OR Asse_J_InFinestraDiPassMode)*) AND
					//Programma_X[X_PosStartLentaDepositoLastra].Stato = TERMINATO (*OR Asse_X_InFinestraDiPassMode)*) AND 
					Programma_Z[Z_PosDepositoInLentaLastra].Stato = TERMINATO (*OR Asse_Z_InFinestraDiPassMode)*) THEN
						Ciclo^.Passo := 90;
						STEPDone := TRUE;
				ELSIF //Programma_Y[Y_PosStartLentaDepositoLastra].Stato = INTERROTTO OR 
					//Programma_J[J_PosDepositoLastra].Stato = INTERROTTO OR 
					//Programma_X[X_PosStartLentaDepositoLastra].Stato = INTERROTTO OR
					Programma_Z[Z_PosDepositoInLentaLastra].Stato = INTERROTTO THEN

					Ciclo^.Passo := 57;								
				END_IF
						
			(* Case 90 - Attesa completamento posizionamento di tutti gli assi *)
			90: 
				IF TFStateCodeGet(ModulePinza^.State) = StateError THEN
					Ciclo^.Passo := 90;																
				ELSE
					RichiestaDepositoALinea := TRUE;
					IF StepInto AND OkDepositoDaLinea THEN
						TFParametersArrayClear(ADR(ParametersArray));
						TFCommandSend(CmdUNLOAD,ParametersArray,ModulePinza^.Cmd);
						Ciclo^.Passo := 91;
						STEPDone := FALSE;
					END_IF							
				END_IF

			(* Case 91 - Attesa completamento rilascio pezzo *)	
			91:
				IF TFStateCodeGet(ModulePinza^.State) = StateError THEN
					Ciclo^.Passo := 91;																
				ELSE
					STEPDone := TRUE;
					IF TFStateCodeGet(ModulePinza^.State) = StateUNLOAD_END THEN//Pezzo rilasciato
						RichiestaDepositoALinea := FALSE;
						Ciclo^.Passo := 92;//dichiaro il ciclo terminato
					END_IF	
				END_IF

			(* Case 92 - Vado in Fuori Ingombro con Z *)
			92:
				IF StepInto then//AND OkDepositoDaLinea THEN
					Programma_Z[Z_PosPostScarico].Stato 			:= DA_ESEGUIRE;
					Programma_Z[Z_PosPostScarico].InterpolaAsse 	:= NO_INTERPOLAZIONE_ASSE;
					ProgrammaToModule_Z 							:= Programma_Z[Z_PosPostScarico];
					Ciclo^.Passo := 93;
					STEPDone := FALSE;
				END_IF

			(* Case 93 - Attesa completamento del comando MOVETOPOS o del raggiungimento quota di Pre-Movimento se abilitata la funzione*)
			93: 
				IF Programma_Z[Z_PosPostScarico].Stato = TERMINATO THEN //OR
				//	Asse_Z_InFinestraDiPassMode OR 
				//	QuotaAnticipoDinamicaZ_Raggiunta THEN
					MaterialeDepositatoSuLinea := TRUE;
					Ciclo^.Passo := 1000;
					STEPDone := TRUE;
				ELSIF Programma_Z[Z_PosPostScarico].Stato = INTERROTTO THEN
					Ciclo^.Passo := 93;										
				END_IF

			(* Case 1000 *)
			1000:
				RichiestaDepositoALinea := FALSE;
				StopDepositoPerArresto := FALSE;
				Ciclo^.Stato := TERMINATO;
				Ciclo^.Passo := 1000;
				
			(* Case 9999 - Ciclo NON annullato o NON terminato*)
			9999:
				Ciclo^.Stato := INTERROTTO;
				Ciclo^.Passo := 9999;
	ELSE						
		;
			
	END_CASE;
ELSE								//Se il ciclo deve essere interrotto, setto il suo nuovo stato
	Ciclo^.Stato := INTERROTTO;
END_IF

END_FUNCTION_BLOCK

// ---- POUs/TFCicliDiLavoro/Lastre/Cicli Depallettizzatore/TFCiclo_Deposito_Falda_Depal.TcPOU
FUNCTION_BLOCK TFCiclo_Deposito_Falda_Depal
VAR_INPUT
	Ciclo 		: POINTER TO Stato_Ciclo_Lavoro;
	Programma  : POINTER TO TFProgramma_Ciclo_Falda_Lastre;
	ModuleAX_X : POINTER TO TFModulePalletizer_Ax;
	ModuleAX_Y : POINTER TO TFModulePalletizer_Ax;
	ModuleAX_Z : POINTER TO TFModulePalletizer_Ax;
	ModuleAX_J : POINTER TO TFModulePalletizer_AxJ_Lastre;
	StartInterpolazioneAssi : POINTER TO BOOL;
	//QuotaPassModePuntoIntermedio : ARRAY [1..3] OF REAL;
	ModulePinza : POINTER TO TFModulePalletizer_Pinza;
	TipoDiDeposito : UINT;
	AbilitazioneGlobalePassMode	: BOOL;
	InterrompiCiclo : BOOL;
	Abilita_Ciclo_Step : BOOL;
	Command_Step : BOOL;
	AbilitazioneAnticipoDinamicoMovimenti : BOOL;
END_VAR
VAR_OUTPUT
	STEPDone	: BOOL;
END_VAR
VAR
	StepInto: BOOL;
END_VAR

(* Set della variabile che mi permette di fare lo STEP nel ciclo *)
StepInto := (Abilita_Ciclo_Step AND Command_Step) OR NOT Abilita_Ciclo_Step;

(* Reset Anticipo Dinamico se non ho l'abilitazione *)
IF NOT AbilitazioneAnticipoDinamicoMovimenti  OR NOT HMI_DisabilitaAnticipiGLOBALE THEN
	QuotaAnticipoDinamicaX_Raggiunta := FALSE;
	QuotaAnticipoDinamicaY_Raggiunta := FALSE;
	QuotaAnticipoDinamicaZ_Raggiunta := FALSE;
END_IF

IF NOT InterrompiCiclo THEN
	IF Ciclo^.Stato = TERMINATO OR Ciclo^.Stato = ANNULLATO THEN
		Ciclo^.Passo := 0;
	ELSIF Ciclo^.Stato = INTERROTTO THEN
		Ciclo^.Passo := 999;
	END_IF
	Ciclo^.Stato := IN_ESECUZIONE;
	CASE Ciclo^.Passo OF
	(* Case 0 *)
			0:  Ciclo^.Stato := IN_ESECUZIONE;
				Ciclo^.Passo := 10;
				STEPDone := FALSE;
		
			(* Case 10 - *)	
			10:	
				Ciclo^.Passo := 11;
				
			(* Case 11 - *)
			11: 
				Ciclo^.Passo := 20;
				
			(* Case 20 - PROGRAMMA[54] ASSE Z -> TRASLAZIONE A QUOTA DI FUORI INGOMBRO *)	
			20:	Ciclo^.Stato := IN_ESECUZIONE;
				IF StepInto THEN
					Programma_Z[Z_PosFuoriIngombroFalda].Stato := DA_ESEGUIRE;
					Programma_Z[Z_PosFuoriIngombroFalda].InterpolaAsse := NO_INTERPOLAZIONE_ASSE;//FALSE;//NO_INTERPOLAZIONE_ASSE
					ProgrammaToModule_Z := Programma_Z[Z_PosFuoriIngombroFalda];
					Ciclo^.Passo := 21;
					STEPDone := FALSE;
				END_IF
				
			(* Case 21 - Attesa completamento del comando MOVETOPOS o del raggiungimento quota di Pre-Movimento se abilitata la funzione *)
			21: 
				IF Programma_Z[Z_PosFuoriIngombroFalda].Stato = TERMINATO OR 
					Asse_Z_InFinestraDiPassMode OR 
					QuotaAnticipoDinamicaZ_Raggiunta THEN
						Ciclo^.Passo := 22;
						STEPDone := TRUE;
				ELSIF Programma_Z[Z_PosFuoriIngombroFalda].Stato = INTERROTTO THEN
					Ciclo^.Passo := 21;										
				END_IF
				
			(* Case 22 - *)
			22:
				Ciclo^.Passo := 23;
				STEPDone := FALSE;
					
			(* Case 23 - *)		
			23:
				Ciclo^.Passo := 24;
				
			(* Case 24 - Scelgo in quale direzione devo muovermi per primo a seconda della disposizione delle postazioni *)	
			24:	
				CASE ASSE_DISPOSIZIONE_POSTAZIONI OF
					
					LUNGO_X:
							Ciclo^.Passo := 25;
				
					LUNGO_Y:	
							IF FuoriIngombroXNecessario THEN
								IF FuoriIngombroYNecessario THEN
									Ciclo^.Passo := 25;
								ELSE
									Ciclo^.Passo := 50;
								END_IF		
							ELSE
								Ciclo^.Passo := 50;
							END_IF
			
				END_CASE
				
			(* Case 25 - Vado a quota di fuori ingombro con Y *)
			25:	IF Programma_Z[Z_PosFuoriIngombroFalda].Stato = INTERROTTO THEN
					Ciclo^.Passo := 25;										
				ELSE
					IF StepInto THEN
						Programma_Y[Y_PosFuoriIngombroVuotoFalda].Stato 			:= DA_ESEGUIRE;
						Programma_Y[Y_PosFuoriIngombroVuotoFalda].InterpolaAsse 	:= NO_INTERPOLAZIONE_ASSE;
						ProgrammaToModule_Y 										:= Programma_Y[Y_PosFuoriIngombroVuotoFalda];
						Ciclo^.Passo := 26;
						STEPDone := FALSE;
					END_IF
				END_IF
					
			(* Case 26 - Check se a quota di fuori ingombro con Y *)		
			26:	IF Programma_Y[Y_PosFuoriIngombroVuotoFalda].Stato = INTERROTTO OR 
					Programma_Z[Z_PosFuoriIngombroFalda].Stato = INTERROTTO THEN
						Ciclo^.Passo := 26;
				ELSE	
					IF Programma_Y[Y_PosFuoriIngombroVuotoFalda].Stato = TERMINATO OR 
						Asse_Y_InFinestraDiPassMode THEN
							Ciclo^.Passo := 30;
							STEPDone := TRUE;							
					END_IF
				END_IF
										
			(* Case 30 - PROGRAMMA[0] ASSE X  -> TRASLAZIONE A QUOTA DI DEPOSITO  *)	
			30:	IF Programma_Z[Z_PosFuoriIngombroFalda].Stato = INTERROTTO OR 
					Programma_Y[Y_PosFuoriIngombroVuotoFalda].Stato = INTERROTTO THEN
						Ciclo^.Passo := 30;										
				ELSE
					IF StepInto THEN
						Programma_X[X_PosDepositoFalda].Stato 			:= DA_ESEGUIRE;
						Programma_X[X_PosDepositoFalda].InterpolaAsse 	:= NO_INTERPOLAZIONE_ASSE;
						ProgrammaToModule_X 							:= Programma_X[X_PosDepositoFalda];
						Ciclo^.Passo := 31;
						STEPDone := FALSE;
					END_IF
				END_IF			
				
			(* Case 31 -  Attesa completamento del comando MOVETOPOS o del raggiungimento quota di Pre-Movimento se abilitata la funzione *)
			31: 
				IF Programma_X[X_PosDepositoFalda].Stato = INTERROTTO OR
					Programma_Y[Y_PosFuoriIngombroVuotoFalda].Stato = INTERROTTO OR
					Programma_Z[Z_PosFuoriIngombroFalda].Stato = INTERROTTO THEN
						Ciclo^.Passo := 31;
				ELSE	
					IF (Programma_X[X_PosDepositoFalda].Stato = TERMINATO OR Asse_X_InFinestraDiPassMode OR QuotaAnticipoDinamicaX_Raggiunta) THEN 
						Ciclo^.Passo := 32;
						STEPDone := TRUE;							
					END_IF
				END_IF
				
			(* Case 32 - Vado a quota di START LENTA CON GLI ASSI con Y,Z,J *)
			32:
				IF Programma_X[X_PosDepositoFalda].Stato = INTERROTTO OR
					Programma_Y[Y_PosFuoriIngombroVuotoFalda].Stato = INTERROTTO OR
					Programma_Z[Z_PosFuoriIngombroFalda].Stato = INTERROTTO THEN
						Ciclo^.Passo := 32;										
				ELSE
					IF StepInto THEN
						TFParametersArrayClear(ADR(ParametersArray));
						Programma_Y[Y_PosDepositoFalda].Stato 			:= DA_ESEGUIRE;
						Programma_Y[Y_PosDepositoFalda].InterpolaAsse 	:= INTERPOLAZIONE_ASSE;
						ProgrammaToModule_Y 							:= Programma_Y[Y_PosDepositoFalda];
				
						//Programma_Z[Z_PosStartLentaDepositoLastra].Stato 			:= DA_ESEGUIRE;
						//Programma_Z[Z_PosStartLentaDepositoLastra].InterpolaAsse 	:= INTERPOLAZIONE_ASSE;
						//ProgrammaToModule_Z 										:= Programma_Z[Z_PosStartLentaDepositoLastra];
						
						Programma_J[J_PosDepositoFalda].Stato 						:= DA_ESEGUIRE;
						Programma_J[J_PosDepositoFalda].InterpolaAsse 				:= INTERPOLAZIONE_ASSE;
						ProgrammaToModule_J 										:= Programma_J[J_PosDepositoFalda];
						
						StartInterpolazioneAssi^ := TRUE; //Abilito l'interpolazione degli assi
												
						Ciclo^.Passo := 33;
						STEPDone := FALSE;
					END_IF
				END_IF
			
			(* Case 33 - Attendo completamento comando o assi in finsetra *)
			33:
				IF (Programma_X[X_PosDepositoFalda].Stato = TERMINATO OR Asse_X_InFinestraDiPassMode OR QuotaAnticipoDinamicaX_Raggiunta) AND
					(Programma_Y[Y_PosDepositoFalda].Stato = TERMINATO OR Asse_Y_InFinestraDiPassMode OR QuotaAnticipoDinamicaY_Raggiunta) AND
					(Programma_J[J_PosDepositoFalda].Stato = TERMINATO OR Asse_J_InFinestraDiPassMode OR QuotaAnticipoDinamicaJ_Raggiunta) THEN
						Ciclo^.Passo := 34;
						STEPDone := TRUE;
				ELSIF Programma_X[X_PosDepositoFalda].Stato = INTERROTTO OR
						Programma_Y[Y_PosDepositoFalda].Stato = INTERROTTO OR 
						Programma_J[J_PosDepositoFalda].Stato = INTERROTTO THEN
							Ciclo^.Passo := 33;								
				END_IF

			(* Case 34 - Vado a quota di finale con Z *)
			34:
				IF Programma_X[X_PosDepositoFalda].Stato = INTERROTTO OR
					Programma_Y[Y_PosDepositoFalda].Stato = INTERROTTO OR
					Programma_J[J_PosDepositoFalda].Stato = INTERROTTO THEN
						Ciclo^.Passo := 34;										
				ELSE
					IF StepInto THEN
						TFParametersArrayClear(ADR(ParametersArray));
				
						Programma_Z[Z_PosStartLentaDepositoFalda].Stato 			:= DA_ESEGUIRE;
						Programma_Z[Z_PosStartLentaDepositoFalda].InterpolaAsse 	:= INTERPOLAZIONE_ASSE;
						ProgrammaToModule_Z 													:= Programma_Z[Z_PosStartLentaDepositoFalda];
												
						StartInterpolazioneAssi^ := TRUE; //Abilito l'interpolazione degli assi
												
						Ciclo^.Passo := 35;
						STEPDone := FALSE;
					END_IF
				END_IF

			(* Case 35 - Attendo completamento comando o assi in finsetra *)
			35:
				IF //Programma_Y[Y_PosStartLentaDepositoLastra].Stato = TERMINATO (*OR Asse_Y_InFinestraDiPassMode)*) AND 
					//Programma_J[J_PosDepositoLastra].Stato = TERMINATO (*OR Asse_J_InFinestraDiPassMode)*) AND
					//Programma_X[X_PosStartLentaDepositoLastra].Stato = TERMINATO (*OR Asse_X_InFinestraDiPassMode)*) AND 
					Programma_Z[Z_PosStartLentaDepositoFalda].Stato = TERMINATO (*OR Asse_Z_InFinestraDiPassMode)*) THEN
						Ciclo^.Passo := 90;
						STEPDone := TRUE;
				ELSIF //Programma_Y[Y_PosStartLentaDepositoLastra].Stato = INTERROTTO OR 
					//Programma_J[J_PosDepositoLastra].Stato = INTERROTTO OR 
					//Programma_X[X_PosStartLentaDepositoLastra].Stato = INTERROTTO OR
					Programma_Z[Z_PosStartLentaDepositoFalda].Stato = INTERROTTO THEN
						Ciclo^.Passo := 35;								
				END_IF
										
			(* Case 50 - Vado a quota di fuori ingombro con X *)
			50:	IF Programma_Z[Z_PosFuoriIngombroFalda].Stato = INTERROTTO THEN
						Ciclo^.Passo := 50;										
				ELSE
					IF StepInto THEN
						Programma_X[X_PosDepositoFalda].Stato 			:= DA_ESEGUIRE;
						Programma_X[X_PosDepositoFalda].InterpolaAsse 	:= NO_INTERPOLAZIONE_ASSE;
						ProgrammaToModule_X 										:= Programma_X[X_PosDepositoFalda];
						Ciclo^.Passo := 51;
						STEPDone := FALSE;
					END_IF
				END_IF
					
			(* Case 51 - Check se a quota di fuori ingombro con Y *)		
			51:	IF Programma_X[X_PosDepositoFalda].Stato = INTERROTTO OR 
					Programma_Z[Z_PosFuoriIngombroFalda].Stato = INTERROTTO THEN
						Ciclo^.Passo := 51;
				ELSE	
					IF Programma_X[X_PosDepositoFalda].Stato = TERMINATO OR 
						Asse_X_InFinestraDiPassMode THEN
							Ciclo^.Passo := 52;
							STEPDone := TRUE;							
					END_IF
				END_IF
										
			(* Case 52 - lancio posizionamento Y+J e X se non serve il fuori ingombro  *)	
			52:	IF Programma_Z[Z_PosFuoriIngombroFalda].Stato = INTERROTTO OR 
					(Programma_X[X_PosDepositoFalda].Stato = INTERROTTO AND FuoriIngombroXNecessario) THEN
						Ciclo^.Passo := 52;										
				ELSE
					IF StepInto THEN
			
					//	IF NOT FuoriIngombroXNecessario THEN
						//	Programma_X[X_PosDepositoSuPostazioneFalda].Stato 			:= DA_ESEGUIRE;
						//	Programma_X[X_PosDepositoSuPostazioneFalda].InterpolaAsse 	:= INTERPOLAZIONE_ASSE;
						//	ProgrammaToModule_X 										:= Programma_X[X_PosDepositoSuPostazioneFalda];
					//	END_IF
					
						Programma_Y[Y_PosDepositoFalda].Stato 			:= DA_ESEGUIRE;
						Programma_Y[Y_PosDepositoFalda].InterpolaAsse 	:= INTERPOLAZIONE_ASSE;
						ProgrammaToModule_Y 										:= Programma_Y[Y_PosDepositoFalda];
						
						//Programma_Z[Z_PosStartLentaDepositoLastra].Stato 			:= DA_ESEGUIRE;
						//Programma_Z[Z_PosStartLentaDepositoLastra].InterpolaAsse 	:= INTERPOLAZIONE_ASSE;
						//ProgrammaToModule_Z 										:= Programma_Z[Z_PosStartLentaDepositoLastra];
					
						Programma_J[J_PosDepositoFalda].Stato 						:= DA_ESEGUIRE;
						Programma_J[J_PosDepositoFalda].InterpolaAsse 				:= INTERPOLAZIONE_ASSE;
						ProgrammaToModule_J 										:= Programma_J[J_PosDepositoFalda];
			
						StartInterpolazioneAssi^ := TRUE; //Abilito l'interpolazione degli assi

						Ciclo^.Passo := 53;
						STEPDone := FALSE;
					END_IF
				END_IF			
				
			(* Case 53 -  Attesa completamento del comando MOVETOPOS o del raggiungimento quota di Pre-Movimento se abilitata la funzione *)
			53: 
				IF Programma_X[X_PosDepositoFalda].Stato = INTERROTTO OR
					Programma_Y[Y_PosDepositoFalda].Stato = INTERROTTO OR
					Programma_Z[Z_PosFuoriIngombroFalda].Stato = INTERROTTO OR 
					Programma_J[J_PosDepositoFalda].Stato = INTERROTTO THEN
						Ciclo^.Passo := 53;
				ELSE	
					IF (Programma_Y[Y_PosDepositoFalda].Stato = TERMINATO OR Asse_Y_InFinestraDiPassMode OR QuotaAnticipoDinamicaY_Raggiunta) AND
						(Programma_J[J_PosDepositoFalda].Stato = TERMINATO OR Asse_J_InFinestraDiPassMode OR QuotaAnticipoDinamicaJ_Raggiunta)  THEN 	
							Ciclo^.Passo := 54;
							STEPDone := TRUE;							
					END_IF
				END_IF
				
			(* Case 54 - Vado a quota di START LENTA CON GLI ASSI Z*)
			54:
				IF Programma_X[X_PosDepositoFalda].Stato 	= INTERROTTO OR
					Programma_Y[Y_PosDepositoFalda].Stato 	= INTERROTTO OR
					Programma_Z[Z_PosFuoriIngombroFalda].Stato 	= INTERROTTO OR 
					Programma_J[J_PosDepositoFalda].Stato 				= INTERROTTO THEN
						Ciclo^.Passo := 54;										
				ELSE
					IF StepInto THEN
						Programma_Z[Z_PosStartLentaDepositoFalda].Stato 			:= DA_ESEGUIRE;
						Programma_Z[Z_PosStartLentaDepositoFalda].InterpolaAsse 	:= NO_INTERPOLAZIONE_ASSE;
						ProgrammaToModule_Z 										:= Programma_Z[Z_PosStartLentaDepositoFalda];
								
						Ciclo^.Passo := 55;
						STEPDone := FALSE;
					END_IF
				END_IF
			
			(* Case 55 - Attendo completamento comando o assi in finsetra *)
			55:
				IF Programma_Y[Y_PosDepositoFalda].Stato = TERMINATO (*OR Asse_Y_InFinestraDiPassMode)*) AND 
					Programma_J[J_PosDepositoFalda].Stato = TERMINATO (*OR Asse_J_InFinestraDiPassMode)*) AND
					Programma_X[X_PosDepositoFalda].Stato = TERMINATO (*OR Asse_X_InFinestraDiPassMode)*) AND 
					Programma_Z[Z_PosStartLentaDepositoFalda].Stato = TERMINATO OR Asse_Z_InFinestraDiPassMode THEN
						Ciclo^.Passo := 56;
						STEPDone := TRUE;
				ELSIF Programma_X[X_PosDepositoFalda].Stato 	= INTERROTTO OR
					Programma_Y[Y_PosDepositoFalda].Stato 	= INTERROTTO OR
					Programma_Z[Z_PosStartLentaDepositoFalda].Stato 	= INTERROTTO OR 
					Programma_J[J_PosDepositoFalda].Stato 				= INTERROTTO THEN
						Ciclo^.Passo := 55;
				END_IF

			(* Case 56 - Vado a quota di finale con Y,Z,J *)
			56:
				IF Programma_X[X_PosStartLentaDepositoLastra].Stato = INTERROTTO OR
					Programma_Y[Y_PosFuoriIngombroCaricoLastra].Stato = INTERROTTO OR
					Programma_Z[Z_PosFuoriIngombroCaricoLastra].Stato = INTERROTTO OR 
					Programma_J[J_PosFuoriIngombro].Stato = INTERROTTO THEN
						Ciclo^.Passo := 56;										
				ELSE
					IF StepInto THEN
						TFParametersArrayClear(ADR(ParametersArray));
						Programma_Z[Z_PosStartLentaDepositoFalda].Stato 			:= DA_ESEGUIRE;
						Programma_Z[Z_PosStartLentaDepositoFalda].InterpolaAsse 	:= NO_INTERPOLAZIONE_ASSE;
						ProgrammaToModule_Z 										:= Programma_Z[Z_PosStartLentaDepositoFalda];						
						Ciclo^.Passo := 57;
						STEPDone := FALSE;
					END_IF
				END_IF

			(* Case 57 - Attendo completamento comando o assi in finsetra *)
			57:
				IF Programma_Z[Z_PosStartLentaDepositoFalda].Stato = TERMINATO (*OR Asse_Z_InFinestraDiPassMode)*) THEN
					Ciclo^.Passo := 90;
					STEPDone := TRUE;
				ELSIF Programma_Z[Z_PosStartLentaDepositoFalda].Stato = INTERROTTO THEN
					Ciclo^.Passo := 57;								
				END_IF
						
			(* Case 90 - Attesa completamento posizionamento di tutti gli assi *)
			90: 
				IF TFStateCodeGet(ModulePinza^.State) = StateError THEN
					Ciclo^.Passo := 90;																
				ELSE
					IF StepInto THEN
						TFParametersArrayClear(ADR(ParametersArray));
						TFCommandSend(CmdUNLOAD,ParametersArray,ModulePinza^.Cmd);
						Ciclo^.Passo := 91;
						STEPDone := FALSE;
					END_IF							
				END_IF

			(* Case 91 - Attesa completamento rilascio pezzo *)	
			91:
				IF TFStateCodeGet(ModulePinza^.State) = StateError THEN
					Ciclo^.Passo := 91;																
				ELSE
					STEPDone := TRUE;
					IF TFStateCodeGet(ModulePinza^.State) = StateUNLOAD_END THEN//Pezzo rilasciato
						Ciclo^.Passo := 1000;//dichiaro il ciclo terminato
					END_IF	
				END_IF

			(* Case 1000 *)
			1000:
				Ciclo^.Stato := TERMINATO;
				Ciclo^.Passo := 1000;
				
			(* Case 9999 - Ciclo NON annullato o NON terminato*)
			9999:
				Ciclo^.Stato := INTERROTTO;
				Ciclo^.Passo := 9999;
	ELSE						
		;
			
	END_CASE;
ELSE								//Se il ciclo deve essere interrotto, setto il suo nuovo stato
	Ciclo^.Stato := INTERROTTO;
END_IF

END_FUNCTION_BLOCK

// ---- POUs/TFPalletizerDataTF/Utility Varie/TFCalcoloTraiettoriaLastre.TcPOU
FUNCTION_BLOCK TFCalcoloTraiettoriaLastre
VAR_INPUT
	Traiettoria : POINTER TO TFTraiettoria;
	WorkSpace : POINTER TO TFMachinePalletizer_WorkSpace;
	WorkFootprint : POINTER TO ARRAY [1..MAXFOOTPRINT] OF TFMachinePalletizer_WorkFootprint;
	WorkPickPoint : POINTER TO ARRAY [1..MAXPICKPOINT] OF TFMachinePalletizer_WorkPickPointSlab;
	WorkPickPointState : POINTER TO ARRAY [1..MAXPICKPOINT] OF TFMachinePalletizer_WorkPickPoint_State;
	WorkPickPointDimension 		: POINTER TO ARRAY [1..MAXPICKPOINT] OF Work_PickPoint_Dimension;

	WorkArea : POINTER TO ARRAY [1..MAXAREA] OF TFMachinePalletizer_WorkArea;
	WorkAreaState : POINTER TO ARRAY [1..MAXAREA] OF TFMachinePalletizer_WorkAreaState;
	Pallet : POINTER TO ARRAY [1..MAXPALLET] OF TFMachinePalletizer_Pallet;
	Layer : POINTER TO ARRAY [1..MAXLAYER] OF TFMachinePalletizer_Layer;
	Forming : POINTER TO ARRAY [1..MAXFORMING] OF TFMachinePalletizer_FormingForSlab;
	//ZDim : REAL;
	
	Mission : POINTER TO TFMachinePalletizer_Mission;
	
	WorkAreaManager : POINTER TO TFWorkAreaManager;
	ModuleAX_X : POINTER TO TFModulePalletizer_Ax;
	ModuleAX_Y : POINTER TO TFModulePalletizer_Ax;
	ModuleAX_Z : POINTER TO TFModulePalletizer_Ax;
	ModuleAX_J : POINTER TO TFModulePalletizer_AxJ_Lastre;
	//ModuleAX_K : POINTER TO TFModulePalletizer_Ax;
	Eseguito : BOOL;
	
END_VAR
VAR
	f : UINT;
	wa : UINT;
	P : UINT;
	a : uint;
	
	WASX : UINT;
	WADX : UINT;
	WAPARTENZA : UINT;
	WADESTINAZIONE : UINT;

	AltezzaDiIngombroArea_CCENTRALE : LREAL; //Altezza ingombro dell'Area nel corridoio CENTRALE
	AltezzaDiIngombroArea_CESTERNO : LREAL; //Altezza ingombro dell'Area nel corridoio ESTERNO
	AltezzaDiIngombroArea_CINTERNO : LREAL; //Altezza ingombro dell'Area nel corridoio INTERNO
	
	AltezzaDiIngombroIngombri_CCENTRALE : LREAL; //Altezza ingombro dell'Area nel corridoio CENTRALE
	AltezzaDiIngombroIngombri_CESTERNO : LREAL; //Altezza ingombro dell'Area nel corridoio ESTERNO
	AltezzaDiIngombroIngombri_CINTERNO : LREAL; //Altezza ingombro dell'Area nel corridoio INTERNO
	

	
	
	AltezzaDiIngombroOstacoli : LREAL;
	AltezzaDiIngombroPuntiPrelievo : LREAL;
	AssegnaQuote : BOOL;
	OffsetSicurezzaConPacco : REAL;
	AltezzaPinzaDaTastatoreAFlangiaMotore : REAL; // Altezza della pinza dal tastatore al bordo superiore della flangia di supporto motore asse K
	AltezzaDaPavimentoAPiastraSupportoColonnaCentrale : REAL;
	LarghezzaPiastraSupportoColonnaCentrale : REAL;
	Quota_X_CentroColonnaCentrale : REAL;
	
	


	(*
	IngombroX_Pos 	: LREAL;//Ingombro della pinza nella Metà POSITIVA della pinza lungo X
	IngombroY_Pos 	: LREAL;//Ingombro della pinza nella Metà POSITIVA della pinza lungo Y
	IngombroZ_Pos 	: LREAL;//Ingombro della pinza nella Metà POSITIVA della pinza lungo Z
	
	IngombroX_Neg 	: LREAL;//Ingombro della pinza nella Metà NEGATIVA della pinza lungo X
	IngombroY_Neg 	: LREAL;//Ingombro della pinza nella Metà NEGATIVA della pinza lungo Y
	IngombroZ_Neg 	: LREAL;//Ingombro della pinza nella Metà NEGATIVA della pinza lungo Z

	IngombroY_Tot 	: LREAL;//Ingombro totale In direzione Y
	*)
	debug : bool;
	CalcolaQuote : BOOL;
	AbilitaValutazioneFISuSingolaWA 		: BOOL;
	NumeroWAValutazioneFISingolaPostazione 	: UINT;
	//TFCalcolaNumeroPostazioneDXSX : TFCalcolaNumeroPostazioneDXSX;
	

END_VAR

(*(* Calcolo gli ingombri della pinza nelle varie direzioni *)
TFCalcoliIngombroPinza(Mission := Mission,
					WorkAreaManager := WorkAreaManager,
					ModuleAX_J := ModuleAX_J,
					AngoloRotazioneDestinazionePinza:= Mission^.JPick,
					IngombroX_Pos := ADR(IngombroX_Pos),
					IngombroY_Pos := ADR(IngombroY_Pos),
					IngombroX_Neg := ADR(IngombroX_Neg),
					IngombroY_Neg := ADR(IngombroY_Neg),
					IngombroZ_Pos := ADR(IngombroZ_Pos),
					IngombroZ_Neg := ADR(IngombroZ_Neg),
					IngombroY_Tot := ADR(IngombroY_Tot),
					IngombroDestinazioneX_Pos := ADR(IngombroDestinazioneX_Pos),
					IngombroDestinazioneY_Pos := ADR(IngombroDestinazioneY_Pos),
					IngombroDestinazioneX_Neg := ADR(IngombroDestinazioneX_Neg),
					IngombroDestinazioneY_Neg := ADR(IngombroDestinazioneY_Neg),
					IngombroDestinazioneZ_Pos := ADR(IngombroDestinazioneZ_Pos),
					IngombroDestinazioneZ_Neg := ADR(IngombroDestinazioneZ_Neg),
					IngombroMaxX_Pos := ADR(IngombroMaxX_Pos),
					IngombroMaxY_Pos := ADR(IngombroMaxY_Pos),
					IngombroMaxX_Neg := ADR(IngombroMaxX_Neg),
					IngombroMaxY_Neg := ADR(IngombroMaxY_Neg),
					IngombroMaxZ_Pos := ADR(IngombroMaxZ_Pos),
					IngombroMaxZ_Neg := ADR(IngombroMaxZ_Neg));*)

CASE WorkAreaManager^.State OF
	WAMANAGER_NOP:
		CalcolaQuote := TRUE;
	
	WAMANAGER_CICLO_RIPOSO_INIT:
		CalcolaQuote := TRUE;

{Region "Ciclo Riposo"}		
	WAMANAGER_CICLO_RIPOSO_RUN:

		IF CalcolaQuote THEN
			CalcolaQuote := FALSE;
			(*QuotaFuoriIngombro_Z_AVUOTO_CCENTRALE 	:= 0;
			QuotaFuoriIngombro_Z_AVUOTO_CESTERNO 	:= 0;
			QuotaFuoriIngombro_Z_AVUOTO_CINTERNO 	:= 0;
			AltezzaDiIngombroPuntiPrelievo := 0;
			AltezzaDiIngombroIngombri_CCENTRALE := 0;
			(* Valuto gli ostacoli *)	
			FOR f:=1 TO MAXFOOTPRINT DO
				AltezzaDiIngombroIngombri_CCENTRALE := MAX(AltezzaDiIngombroIngombri_CCENTRALE,WorkFootPrint^[f].Z + WorkFootPrint^[f].ZDim + IngombroMaxZ_Neg);
			END_FOR

			(* Valuto I Pick-Point *)
			FOR P:=1 TO MAXPICKPOINT DO	
				AltezzaDiIngombroPuntiPrelievo := MAX(AltezzaDiIngombroPuntiPrelievo,WorkPickPointDimension^[P].Zdim,WorkPickPoint^[P].ZRaise,WorkPickPoint^[P].Z);
			END_FOR

			(* Valuto le wa *)			
			CASE ASSE_DISPOSIZIONE_POSTAZIONI OF
				
				LUNGO_X:
						CalcolaIngombroWALungoX_Pal();
				
				LUNGO_Y:
						CalcolaIngombroWALungoY_Pal();
			
			END_CASE

			QuotaFuoriIngombro_Z_AVUOTO_CCENTRALE := MAX(AltezzaDiIngombroArea_CCENTRALE,AltezzaDiIngombroIngombri_CCENTRALE,AltezzaDiIngombroPuntiPrelievo) + IngombroMaxZ_Neg;
			QuotaFuoriIngombro_Z_AVUOTO_CESTERNO := MAX(AltezzaDiIngombroArea_CESTERNO,AltezzaDiIngombroIngombri_CCENTRALE,AltezzaDiIngombroPuntiPrelievo) + IngombroMaxZ_Neg;
			QuotaFuoriIngombro_Z_AVUOTO_CINTERNO := MAX(AltezzaDiIngombroArea_CINTERNO,AltezzaDiIngombroIngombri_CCENTRALE,AltezzaDiIngombroPuntiPrelievo) +IngombroMaxZ_Neg;
			QuotaFuoriIngombro_Z_AVUOTO := MAX(QuotaFuoriIngombro_Z_AVUOTO_CCENTRALE,QuotaFuoriIngombro_Z_AVUOTO_CESTERNO,QuotaFuoriIngombro_Z_AVUOTO_CINTERNO)+OffsetSicurezza.Z.Avuoto;
			*)
			(* Valuto se gli assi sono in finestra di prelievo, in questo modo valuto nel ciclo se devo andare fuori ingombro oppure posso partire da dove sono *)
			AsseXInFinestraDiPrelievo := FALSE;
			IF (ModuleAx_X^.Ax^.AxRef^.NcToPlc.ActPos >= Mission^.XPick - 50) AND (ModuleAx_X^.Ax^.AxRef^.NcToPlc.ActPos <=  Mission^.XPick + 50) THEN
				AsseXInFinestraDiPrelievo := TRUE;
			END_IF
			AsseYInFinestraDiPrelievo := FALSE;
			IF (ModuleAx_Y^.Ax^.AxRef^.NcToPlc.ActPos  >=  Mission^.YPick - 50) AND (ModuleAx_Y^.Ax^.AxRef^.NcToPlc.SetPos <= Mission^.YPick + 50) THEN
				AsseYInFinestraDiPrelievo := TRUE;
			END_IF
			(* Valuto la rotazione della pinza *)
			AsseJInFinestraDiPrelievo := FALSE;
			IF ModuleAx_J^.Ax^.AxRef^.NcToPlc.ActPos >= Mission^.JPick - 5 AND ModuleAx_J^.Ax^.AxRef^.NcToPlc.ActPos <= Mission^.JPick + 5 THEN
				AsseJInFinestraDiPrelievo := TRUE;
			END_IF
			
		END_IF

		//QuotaFuoriIngombro_Z_AVUOTO := MAX(QuotaFuoriIngombro_Z_AVUOTO_CCENTRALE,QuotaFuoriIngombro_Z_AVUOTO_CESTERNO,QuotaFuoriIngombro_Z_AVUOTO_CINTERNO)+OffsetSicurezza.Z.Avuoto;
		//QuotaFuoriIngombro_Z_ConPEZZO := MAX(QuotaFuoriIngombro_Z_AVUOTO_CCENTRALE,QuotaFuoriIngombro_Z_AVUOTO_CESTERNO,QuotaFuoriIngombro_Z_AVUOTO_CINTERNO)+OffsetSicurezza.Z.Carico;


	WAMANAGER_CICLO_RIPOSO_END:
		CalcolaQuote := TRUE;
{Endregion}

{Region "CCLO LASTRA PP"}
	WAMANAGER_CICLO_LASTRA_PP_INIT:
		CalcolaQuote := TRUE;

	WAMANAGER_CICLO_PRELIEVO_LASTRA_PP_RUN:
		
		IF CalcolaQuote THEN
			(*CalcolaQuote := FALSE;
			QuotaFuoriIngombro_Z_AVUOTO_CCENTRALE 	:= 0;
			QuotaFuoriIngombro_Z_AVUOTO_CESTERNO 	:= 0;
			QuotaFuoriIngombro_Z_AVUOTO_CINTERNO 	:= 0;
			AltezzaDiIngombroPuntiPrelievo := 0;
			AltezzaDiIngombroIngombri_CCENTRALE := 0;
			(* Valuto gli ostacoli *)	
			FOR f:=1 TO MAXFOOTPRINT DO
				AltezzaDiIngombroIngombri_CCENTRALE := MAX(AltezzaDiIngombroIngombri_CCENTRALE,WorkFootPrint^[f].Z + WorkFootPrint^[f].ZDim + IngombroMaxZ_Neg);
			END_FOR

			(* Valuto I Pick-Point *)
			FOR P:=1 TO MAXPICKPOINT DO	
				AltezzaDiIngombroPuntiPrelievo := MAX(AltezzaDiIngombroPuntiPrelievo,WorkPickPointDimension^[P].Zdim,WorkPickPoint^[P].ZRaise,WorkPickPoint^[P].Z);
			END_FOR
			//Per la postazione 2 valuto il FI solo della postazione stessa perchè non è in interferenza con la postazione n°1
			AbilitaValutazioneFISuSingolaWA 		:= FALSE;
			NumeroWAValutazioneFISingolaPostazione 	:= 0;
			//IF Mission^.PPick = 2 THEN
			//	AbilitaValutazioneFISuSingolaWA 		:= TRUE;
			//	NumeroWAValutazioneFISingolaPostazione 	:= 2;
			//END_IF


			(* Valuto le wa *)			
			CASE ASSE_DISPOSIZIONE_POSTAZIONI OF
				
				LUNGO_X:
						CalcolaIngombroWALungoX_Pal();
				
				LUNGO_Y:
						CalcolaIngombroWALungoY_Pal();
			
			END_CASE
	
			QuotaFuoriIngombro_Z_AVUOTO_CCENTRALE := MAX(AltezzaDiIngombroArea_CCENTRALE,AltezzaDiIngombroIngombri_CCENTRALE,AltezzaDiIngombroPuntiPrelievo) + IngombroMaxZ_Neg;
			QuotaFuoriIngombro_Z_AVUOTO_CESTERNO := MAX(AltezzaDiIngombroArea_CESTERNO,AltezzaDiIngombroIngombri_CCENTRALE,AltezzaDiIngombroPuntiPrelievo) + IngombroMaxZ_Neg;
			QuotaFuoriIngombro_Z_AVUOTO_CINTERNO := MAX(AltezzaDiIngombroArea_CINTERNO,AltezzaDiIngombroIngombri_CCENTRALE,AltezzaDiIngombroPuntiPrelievo) +IngombroMaxZ_Neg;
			QuotaFuoriIngombro_Z_AVUOTO := MAX(QuotaFuoriIngombro_Z_AVUOTO_CCENTRALE,QuotaFuoriIngombro_Z_AVUOTO_CESTERNO,QuotaFuoriIngombro_Z_AVUOTO_CINTERNO)+OffsetSicurezza.Z.Avuoto;
			*)	
			(* Valuto se gli assi sono in finestra di prelievo, in questo modo valuto nel ciclo se devo andare fuori ingombro oppure posso partire da dove sono *)
			AsseXInFinestraDiPrelievo := FALSE;
			IF (ModuleAx_X^.Ax^.AxRef^.NcToPlc.ActPos >= Mission^.XPick - 50) AND (ModuleAx_X^.Ax^.AxRef^.NcToPlc.ActPos <=  Mission^.XPick + 50) THEN
				AsseXInFinestraDiPrelievo := TRUE;
			END_IF
			AsseYInFinestraDiPrelievo := FALSE;
			IF (ModuleAx_Y^.Ax^.AxRef^.NcToPlc.ActPos  >=  Mission^.YPick - 50) AND (ModuleAx_Y^.Ax^.AxRef^.NcToPlc.ActPos <= Mission^.YPick + 50) THEN
				AsseYInFinestraDiPrelievo := TRUE;
			END_IF
			(* Valuto la rotazione della pinza *)
			AsseJInFinestraDiPrelievo := FALSE;
			IF ModuleAx_J^.Ax^.AxRef^.NcToPlc.ActPos >= Mission^.JPick - 5 AND ModuleAx_J^.Ax^.AxRef^.NcToPlc.ActPos <= Mission^.JPick + 5 THEN
				AsseJInFinestraDiPrelievo := TRUE;
			END_IF
	
		END_IF //riferito all'IF dello stato della missione	
			
		//QuotaFuoriIngombro_Z_AVUOTO := MAX(QuotaFuoriIngombro_Z_AVUOTO_CCENTRALE,QuotaFuoriIngombro_Z_AVUOTO_CESTERNO,QuotaFuoriIngombro_Z_AVUOTO_CINTERNO)+OffsetSicurezza.Z.Avuoto;
		//QuotaFuoriIngombro_Z_ConPEZZO := MAX(QuotaFuoriIngombro_Z_AVUOTO_CCENTRALE,QuotaFuoriIngombro_Z_AVUOTO_CESTERNO,QuotaFuoriIngombro_Z_AVUOTO_CINTERNO)+OffsetSicurezza.Z.Carico;

		Traiettoria^.PuntoDiPostPosizionamentoStartPoint.Z := Mission^.ZPick + OffsetDistacco.Lastra.Z;
		
		
	WAMANAGER_CICLO_PRELIEVO_LASTRA_PP_END:
		CalcolaQuote := TRUE;

	WAMANAGER_CICLO_DEPOSITO_LASTRA_PP_RUN:

		IF CalcolaQuote THEN
			(*CalcolaQuote := FALSE;

			QuotaFuoriIngombro_Z_AVUOTO_CCENTRALE 	:= 0;
			QuotaFuoriIngombro_Z_AVUOTO_CESTERNO 	:= 0;
			QuotaFuoriIngombro_Z_AVUOTO_CINTERNO 	:= 0;
			AltezzaDiIngombroPuntiPrelievo := 0;
			AltezzaDiIngombroIngombri_CCENTRALE := 0;
			(* Valuto gli ostacoli *)	
			FOR f:=1 TO MAXFOOTPRINT DO
				AltezzaDiIngombroIngombri_CCENTRALE := MAX(AltezzaDiIngombroIngombri_CCENTRALE,WorkFootPrint^[f].Z + WorkFootPrint^[f].ZDim + IngombroMaxZ_Neg);
			END_FOR

			(* Valuto I Pick-Point *)
			FOR P:=1 TO MAXPICKPOINT DO	
				AltezzaDiIngombroPuntiPrelievo := MAX(AltezzaDiIngombroPuntiPrelievo,WorkPickPointDimension^[P].Zdim,WorkPickPoint^[P].ZRaise,WorkPickPoint^[P].Z);
			END_FOR

			//Per la postazione 2 valuto il FI solo della postazione stessa perchè non è in interferenza con la postazione n°1
			AbilitaValutazioneFISuSingolaWA 		:= FALSE;
			NumeroWAValutazioneFISingolaPostazione 	:= 0;
			IF Mission^.PPick = 2 THEN
				AbilitaValutazioneFISuSingolaWA 		:= TRUE;
				NumeroWAValutazioneFISingolaPostazione 	:= 2;
			END_IF
			(* Valuto le wa *)			
			CASE ASSE_DISPOSIZIONE_POSTAZIONI OF
				
				LUNGO_X:
						CalcolaIngombroWALungoX_Pal();
				
				LUNGO_Y:
						CalcolaIngombroWALungoY_Pal();
			
			END_CASE

			QuotaFuoriIngombro_Z_AVUOTO_CCENTRALE := MAX(AltezzaDiIngombroArea_CCENTRALE,AltezzaDiIngombroIngombri_CCENTRALE,AltezzaDiIngombroPuntiPrelievo) + IngombroMaxZ_Neg;
			QuotaFuoriIngombro_Z_AVUOTO_CESTERNO := MAX(AltezzaDiIngombroArea_CESTERNO,AltezzaDiIngombroIngombri_CCENTRALE,AltezzaDiIngombroPuntiPrelievo) + IngombroMaxZ_Neg;
			QuotaFuoriIngombro_Z_AVUOTO_CINTERNO := MAX(AltezzaDiIngombroArea_CINTERNO,AltezzaDiIngombroIngombri_CCENTRALE,AltezzaDiIngombroPuntiPrelievo) +IngombroMaxZ_Neg;
			QuotaFuoriIngombro_Z_AVUOTO := MAX(QuotaFuoriIngombro_Z_AVUOTO_CCENTRALE,QuotaFuoriIngombro_Z_AVUOTO_CESTERNO,QuotaFuoriIngombro_Z_AVUOTO_CINTERNO)+OffsetSicurezza.Z.Avuoto;
	
			(* Valuto se gli assi sono in finestra di prelievo, in questo modo valuto nel ciclo se devo andare fuori ingombro oppure posso partire da dove sono *)
			AsseXInFinestraDiPrelievo := FALSE;
			IF (ModuleAx_X^.Ax^.AxRef^.NcToPlc.ActPos >= Mission^.XPick - 50) AND (ModuleAx_X^.Ax^.AxRef^.NcToPlc.ActPos <=  Mission^.XPick + 50) THEN
				AsseXInFinestraDiPrelievo := TRUE;
			END_IF
			AsseYInFinestraDiPrelievo := FALSE;
			IF (ModuleAx_Y^.Ax^.AxRef^.NcToPlc.ActPos  >=  Mission^.YPick - 50) AND (ModuleAx_Y^.Ax^.AxRef^.NcToPlc.SetPos <= Mission^.YPick + 50) THEN
				AsseYInFinestraDiPrelievo := TRUE;
			END_IF
			(* Valuto la rotazione della pinza *)
			AsseJInFinestraDiPrelievo := FALSE;
			IF ModuleAx_J^.Ax^.AxRef^.NcToPlc.ActPos >= Mission^.JPick - 5 AND ModuleAx_J^.Ax^.AxRef^.NcToPlc.ActPos <= Mission^.JPick + 5 THEN
				AsseJInFinestraDiPrelievo := TRUE;
			END_IF
			FuoriIngombroXNecessario := NOT AsseXInFinestraDiPrelievo;
			FuoriIngombroYNecessario := NOT AsseYInFinestraDiPrelievo;*)
		END_IF

		//QuotaFuoriIngombro_Z_AVUOTO := MAX(QuotaFuoriIngombro_Z_AVUOTO_CCENTRALE,QuotaFuoriIngombro_Z_AVUOTO_CESTERNO,QuotaFuoriIngombro_Z_AVUOTO_CINTERNO)+OffsetSicurezza.Z.Avuoto;
		//QuotaFuoriIngombro_Z_ConPEZZO := MAX(QuotaFuoriIngombro_Z_AVUOTO_CCENTRALE,QuotaFuoriIngombro_Z_AVUOTO_CESTERNO,QuotaFuoriIngombro_Z_AVUOTO_CINTERNO)+OffsetSicurezza.Z.Carico;
	
		Traiettoria^.PuntoDiPostPosizionamentoStartPoint.Z := Mission^.ZPick + OffsetDistacco.Lastra.Z;
		
	WAMANAGER_CICLO_DEPOSITO_LASTRA_PP_END:
		CalcolaQuote := TRUE;
{Endregion}

{Region "CCLO LASTRA WA"}
	WAMANAGER_CICLO_LASTRA_WA_INIT:
		CalcolaQuote := TRUE;

	WAMANAGER_CICLO_PRELIEVO_LASTRA_WA_RUN:
		
		IF CalcolaQuote THEN
			(* Valuto se gli assi sono in finestra di prelievo, in questo modo valuto nel ciclo se devo andare fuori ingombro oppure posso partire da dove sono *)
			AsseXInFinestraDiPrelievo := FALSE;
			IF (ModuleAx_X^.Ax^.AxRef^.NcToPlc.ActPos >= Mission^.XPick - 50) AND (ModuleAx_X^.Ax^.AxRef^.NcToPlc.ActPos <=  Mission^.XPick + 50) THEN
				AsseXInFinestraDiPrelievo := TRUE;
			END_IF
			AsseYInFinestraDiPrelievo := FALSE;
			IF (ModuleAx_Y^.Ax^.AxRef^.NcToPlc.ActPos  >=  Mission^.YPick - 50) AND (ModuleAx_Y^.Ax^.AxRef^.NcToPlc.ActPos <= Mission^.YPick + 50) THEN
				AsseYInFinestraDiPrelievo := TRUE;
			END_IF
			(* Valuto la rotazione della pinza *)
			AsseJInFinestraDiPrelievo := FALSE;
			IF ModuleAx_J^.Ax^.AxRef^.NcToPlc.ActPos >= Mission^.JPick - 5 AND ModuleAx_J^.Ax^.AxRef^.NcToPlc.ActPos <= Mission^.JPick + 5 THEN
				AsseJInFinestraDiPrelievo := TRUE;
			END_IF
			
			Traiettoria^.PuntoDiPostPosizionamentoStartPoint.Z := Mission^.ZPick + OffsetDistacco.Falda.Z;
		END_IF


	WAMANAGER_CICLO_PRELIEVO_LASTRA_WA_END:
		CalcolaQuote := TRUE;

	WAMANAGER_CICLO_DEPOSITO_LASTRA_WA_RUN:

		IF CalcolaQuote THEN
			Traiettoria^.PuntoDiPostPosizionamentoStartPoint.Z := Mission^.ZPick + OffsetDistacco.Falda.Z;
		
		
			IF Mission^.JPlace >= 85 AND Mission^.JPlace <= 95 AND HMI_AbilitaDepositoPaccoOrrizzontaleConTasteggio THEN
				Mission^.ZPlace	:= Mission^.ZPlace -100;
			ELSE
				Mission^.ZPlace := Mission^.ZPlace;
			END_IF
			CalcolaQuote := FALSE;
		END_IF		
		//QuotaFuoriIngombro_Z_AVUOTO := MAX(QuotaFuoriIngombro_Z_AVUOTO_CCENTRALE,QuotaFuoriIngombro_Z_AVUOTO_CESTERNO,QuotaFuoriIngombro_Z_AVUOTO_CINTERNO)+OffsetSicurezza.Z.Avuoto;
		//QuotaFuoriIngombro_Z_ConPEZZO := MAX(QuotaFuoriIngombro_Z_AVUOTO_CCENTRALE,QuotaFuoriIngombro_Z_AVUOTO_CESTERNO,QuotaFuoriIngombro_Z_AVUOTO_CINTERNO)+OffsetSicurezza.Z.Carico;
	
	WAMANAGER_CICLO_DEPOSITO_LASTRA_WA_END:
		CalcolaQuote := TRUE;
{Endregion}

END_CASE

(* Punto di approccio iniziale - Necessario per lo start lenta *)
Traiettoria^.PuntoDiApproccioStartPoint.X := Mission^.XPickApproach;
Traiettoria^.PuntoDiApproccioStartPoint.Y := Mission^.YPickApproach;
Traiettoria^.PuntoDiApproccioStartPoint.Z := Mission^.ZPickApproach;
Traiettoria^.PuntoDiApproccioStartPoint.J := Mission^.JPickApproach;
///////////////////////////////////////////////////////////////////////////////////////////////////////////////////////////////////////////////////////////
///////////////////////////////////////////////////////////////////////////////////////////////////////////////////////////////////////////////////////////

(* Punto iniziale - Cincidente con il punto di prelievo *)
Traiettoria^.StartPoint.X := Mission^.XPick;
Traiettoria^.StartPoint.Y := Mission^.YPick;
Traiettoria^.StartPoint.Z := Mission^.ZPick;// - 100;
Traiettoria^.StartPoint.J := Mission^.JPick;

Traiettoria^.PuntoDiPostPosizionamentoStartPoint.X := Mission^.XPick;
IF Mission^.JPick > 90 THEN		
	Traiettoria^.PuntoDiPostPosizionamentoStartPoint.Y := Mission^.YPick + OffsetDistacco.Lastra.Y;
ELSIF Mission^.JPick < 90 THEN	
	//Traiettoria^.PuntoDiPostPosizionamentoStartPoint.Y := Mission^.YPick - OffsetDistacco.Lastra.Y;
	Traiettoria^.PuntoDiPostPosizionamentoStartPoint.Y := Mission^.YPick - OffsetDistacco.Lastra.Y;
END_IF	
 
Traiettoria^.PuntoDiPostPosizionamentoStartPoint.Z := Mission^.ZPick + OffsetDistacco.Lastra.Z;
Traiettoria^.PuntoDiPostPosizionamentoStartPoint.J := Mission^.JPick;

///////////////////////////////////////////////////////////////////////////////////////////////////////////////////////////////////////////////////////////
///////////////////////////////////////////////////////////////////////////////////////////////////////////////////////////////////////////////////////////
(* Punto di approccio finale :
- nel caso di deposito falda su catasta con apprendimento, la quota Z di approccio coincide con la quota di start lenta
- nel caso di deposito falda su catasta SENZA apprendimento, la quota Z di approccio coincide con la quota di start lenta per evitare che se c'è un pallet fuori sagoma, evitiamo collisioni brusche della pinza*)

Traiettoria^.PuntoDiApproccioEndPoint.X := Mission^.XPlaceApproach;
Traiettoria^.PuntoDiApproccioEndPoint.Y := Mission^.YPlaceApproach;
Traiettoria^.PuntoDiApproccioEndPoint.Z := Mission^.ZPlaceApproach;
Traiettoria^.PuntoDiApproccioEndPoint.J := Mission^.JPlaceApproach;

Traiettoria^.PuntoDiApproccioSecondarioEndPoint.X := Mission^.XPlaceApproachSecondario;
Traiettoria^.PuntoDiApproccioSecondarioEndPoint.Y := Mission^.YPlaceApproachSecondario;
Traiettoria^.PuntoDiApproccioSecondarioEndPoint.Z := Mission^.ZPlaceApproachSecondario;
Traiettoria^.PuntoDiApproccioSecondarioEndPoint.J := Mission^.JPlaceApproachSecondario;

/////////////////////////////////////////////////////////////////////////////////////////////////////////////////////////////////////////////////////////////
/////////////////////////////////////////////////////////////////////////////////////////////////////////////////////////////////////////////////////////////
(* Punto finale*)
Traiettoria^.EndPoint.X := Mission^.XPlace;
Traiettoria^.EndPoint.Y := Mission^.YPlace;
Traiettoria^.EndPoint.Z := Mission^.ZPlace;
Traiettoria^.EndPoint.J := Mission^.JPlace;

Traiettoria^.EndPointSecondario.X := Mission^.XPlaceSecondario;
Traiettoria^.EndPointSecondario.Y := Mission^.YPlaceSecondario;
Traiettoria^.EndPointSecondario.Z := Mission^.ZPlaceSecondario;
Traiettoria^.EndPointSecondario.J := Mission^.JPlaceSecondario;

//
Traiettoria^.PassModeGlobalEnable := AbilitazionePassModeGlobale;

ACTION CalcolaIngombroWALungoX:
/////////////////////////////////////////////////////////////!!!!!!!!!!!!!!!!!!!!!!!!!!!!!!!!//////////////////////////////
(*TFCalcolaNumeroPostazioneDXSX(PosizioneAttuale:=ModuleAX_X^.Ax^.Status.ActPosition,
								WorkArea:=WorkArea,
								DirezioneAsseX_Positiva:= TFDirezioneAssePositiva(Posizione_Attuale:=ModuleAX_X^.Ax^.Status.ActPosition,Posizione_Finale:=Mission^.XPick),
								NPostazioneDX=>WADX,
								NPostazioneSX=>WASX,
								PostazionePartenza=>WAPARTENZA);*)
								
AltezzaDiIngombroArea_CCENTRALE := 0;
AltezzaDiIngombroArea_CESTERNO := 0;
AltezzaDiIngombroArea_CESTERNO := 0;
FOR wa := 1 TO MAXAREAPRESENT DO
	
	CASE WorkArea^[wa].Typology OF
		TYPOLOGY_PALLET:
			CASE WorkAreaState^[wa].TransportState.Supporto.Tipologia OF
					
				PALLET_STANDARD:

					AltezzaDiIngombroArea_CCENTRALE := MAX(AltezzaDiIngombroArea_CCENTRALE, 
															WorkArea^[wa].Z +  MAX(//WorkArea^[wa].Z,
															WorkAreaState^[wa].H,
															WorkAreaState^[wa].HPL,
															WorkAreaState^[wa].TransportState.Supporto.HMAX,
															WorkAreaState^[wa].TransportState.Supporto.ZDim));

					AltezzaDiIngombroArea_CESTERNO	:= AltezzaDiIngombroArea_CCENTRALE;
					AltezzaDiIngombroArea_CINTERNO	:= AltezzaDiIngombroArea_CCENTRALE;
					
				PALLET_ACCOPPIATI:

					AltezzaDiIngombroArea_CCENTRALE := MAX(AltezzaDiIngombroArea_CCENTRALE, 
															WorkArea^[wa].Z +  MAX(//WorkArea^[wa].Z,
															WorkAreaState^[wa].H,
															WorkAreaState^[wa].HPL,
															WorkAreaState^[wa].TransportState.Supporto.HMAX,
															WorkAreaState^[wa].TransportState.Supporto.ZDim));

					AltezzaDiIngombroArea_CESTERNO	:= AltezzaDiIngombroArea_CCENTRALE;
					AltezzaDiIngombroArea_CINTERNO	:= AltezzaDiIngombroArea_CCENTRALE;
					
					
				CASSA_STANDARD:
									
					AltezzaDiIngombroArea_CCENTRALE := MAX(AltezzaDiIngombroArea_CCENTRALE, 
															WorkArea^[wa].Z +  MAX(//WorkArea^[wa].Z,
															WorkAreaState^[wa].H,
															WorkAreaState^[wa].HPL,
															WorkAreaState^[wa].TransportState.Supporto.HMAX,
															WorkAreaState^[wa].TransportState.Supporto.ZDim));

					AltezzaDiIngombroArea_CESTERNO	:= AltezzaDiIngombroArea_CCENTRALE;
					AltezzaDiIngombroArea_CINTERNO	:= AltezzaDiIngombroArea_CCENTRALE;
					
					
				CAVALLETTO:
					AltezzaDiIngombroArea_CCENTRALE := MAX(AltezzaDiIngombroArea_CCENTRALE, 
															WorkArea^[wa].Z,
															WorkAreaState^[wa].TransportState.Supporto.HMAX,
															WorkAreaState^[wa].TransportState.Supporto.ZDim);

					AltezzaDiIngombroArea_CESTERNO	:= MAX(AltezzaDiIngombroArea_CESTERNO,
															WorkArea^[wa].Z,
															//WorkAreaState^[wa].WorkPickPointTransportState.Supporto.HMAX,
															WorkAreaState^[wa].TransportState.Supporto.ZDim);

					AltezzaDiIngombroArea_CINTERNO	:= AltezzaDiIngombroArea_CESTERNO;
				
				BUNDLE:
					AltezzaDiIngombroArea_CCENTRALE := MAX(AltezzaDiIngombroArea_CCENTRALE, 
															WorkArea^[wa].Z,
															WorkAreaState^[wa].TransportState.Supporto.HMAX,
															WorkAreaState^[wa].TransportState.Supporto.ZDim);

					AltezzaDiIngombroArea_CESTERNO	:= MAX(AltezzaDiIngombroArea_CESTERNO,
															WorkArea^[wa].Z,
															//WorkAreaState^[wa].WorkPickPointTransportState.Supporto.HMAX,
															WorkAreaState^[wa].TransportState.Supporto.ZDim);

					AltezzaDiIngombroArea_CINTERNO	:= AltezzaDiIngombroArea_CESTERNO;
					
				ELSE
					AltezzaDiIngombroArea_CCENTRALE := WorkArea^[wa].Z;//Fisso l'altezza ad una quota di default
			END_CASE
						
		TYPOLOGY_LAYER:
			AltezzaDiIngombroArea_CCENTRALE := MAX(AltezzaDiIngombroArea_CCENTRALE,
													WorkArea^[wa].Z,
													WorkAreaState^[wa].H,
													WorkAreaState^[wa].HPL);

			AltezzaDiIngombroArea_CESTERNO	:= AltezzaDiIngombroArea_CCENTRALE;
			AltezzaDiIngombroArea_CINTERNO	:= AltezzaDiIngombroArea_CCENTRALE;
		
		TYPOLOGY_EXTERNAL_DEPPREL:
			AltezzaDiIngombroArea_CCENTRALE := AltezzaDiIngombroArea_CCENTRALE;
					
		TYPOLOGY_OVER_TRANSPORT:
			CASE WorkAreaState^[wa].TransportState.Supporto.Tipologia OF
					
				PALLET_STANDARD:

					AltezzaDiIngombroArea_CCENTRALE := MAX(AltezzaDiIngombroArea_CCENTRALE, 
															WorkArea^[wa].Z +  MAX(//WorkArea^[wa].Z,
															WorkAreaState^[wa].H,
															WorkAreaState^[wa].HPL,
															WorkAreaState^[wa].TransportState.Supporto.HMAX,
															WorkAreaState^[wa].TransportState.Supporto.ZDim));

					AltezzaDiIngombroArea_CESTERNO	:= AltezzaDiIngombroArea_CCENTRALE;
					AltezzaDiIngombroArea_CINTERNO	:= AltezzaDiIngombroArea_CCENTRALE;
					
				PALLET_ACCOPPIATI:

					AltezzaDiIngombroArea_CCENTRALE := MAX(AltezzaDiIngombroArea_CCENTRALE, 
															WorkArea^[wa].Z +  MAX(//WorkArea^[wa].Z,
															WorkAreaState^[wa].H,
															WorkAreaState^[wa].HPL,
															WorkAreaState^[wa].TransportState.Supporto.HMAX,
															WorkAreaState^[wa].TransportState.Supporto.ZDim));

					AltezzaDiIngombroArea_CESTERNO	:= AltezzaDiIngombroArea_CCENTRALE;
					AltezzaDiIngombroArea_CINTERNO	:= AltezzaDiIngombroArea_CCENTRALE;
	
				CASSA_STANDARD:
									
					AltezzaDiIngombroArea_CCENTRALE := MAX(AltezzaDiIngombroArea_CCENTRALE, 
															WorkArea^[wa].Z +  MAX(//WorkArea^[wa].Z,
															WorkAreaState^[wa].H,
															WorkAreaState^[wa].HPL,
															WorkAreaState^[wa].TransportState.Supporto.HMAX,
															WorkAreaState^[wa].TransportState.Supporto.ZDim));

					AltezzaDiIngombroArea_CESTERNO	:= AltezzaDiIngombroArea_CCENTRALE;
					AltezzaDiIngombroArea_CINTERNO	:= AltezzaDiIngombroArea_CCENTRALE;
					
					
				CAVALLETTO:
					AltezzaDiIngombroArea_CCENTRALE := MAX(AltezzaDiIngombroArea_CCENTRALE, 
															WorkArea^[wa].Z,
															WorkAreaState^[wa].TransportState.Supporto.HMAX,
															WorkAreaState^[wa].TransportState.Supporto.ZDim);

					AltezzaDiIngombroArea_CESTERNO	:= MAX(AltezzaDiIngombroArea_CESTERNO,
															WorkArea^[wa].Z,
															//WorkAreaState^[wa].WorkPickPointTransportState.Supporto.HMAX,
															WorkAreaState^[wa].TransportState.Supporto.ZDim);

					AltezzaDiIngombroArea_CINTERNO	:= AltezzaDiIngombroArea_CESTERNO;
				
				BUNDLE:
					AltezzaDiIngombroArea_CCENTRALE := MAX(AltezzaDiIngombroArea_CCENTRALE, 
															WorkArea^[wa].Z,
															WorkAreaState^[wa].TransportState.Supporto.HMAX,
															WorkAreaState^[wa].TransportState.Supporto.ZDim);

					AltezzaDiIngombroArea_CESTERNO	:= MAX(AltezzaDiIngombroArea_CESTERNO,
															WorkArea^[wa].Z,
															//WorkAreaState^[wa].WorkPickPointTransportState.Supporto.HMAX,
															WorkAreaState^[wa].TransportState.Supporto.ZDim);

					AltezzaDiIngombroArea_CINTERNO	:= AltezzaDiIngombroArea_CESTERNO;
				
				ELSE
					AltezzaDiIngombroArea_CCENTRALE := WorkArea^[wa].Z;//Fisso l'altezza ad una quota di default
			END_CASE
	END_CASE															
END_FOR	
		
(*ELSE
	(*TFCalcolaNumeroPostazioneDXSX(PosizioneAttuale	:= ModuleAX_X^.Ax^.Status.ActPosition,
									WorkArea		:= WorkArea,
									DirezioneAsseX_Positiva:=FALSE,
									NPostazioneDX	=> WADX,
									NPostazioneSX	=> WASX,
									PostazionePartenza=>WAPARTENZA);*)
			
	FOR wa := MAXAREA TO 1 BY -1 DO
		AltezzaDiIngombroArea_CCENTRALE := 0;
		IF WorkAreaState^[wa].H > WorkAreaState^[wa].HPL THEN
			AltezzaDiIngombroArea_CCENTRALE := WorkAreaState^[wa].H;
		ELSE
			AltezzaDiIngombroArea_CCENTRALE := WorkAreaState^[wa].HPL;
		END_IF
		IF QuotaFuoriIngombro_Z_AVUOTO_CCENTRALE <= AltezzaDiIngombroArea_CCENTRALE + TCPParameter.Z + OffsetSicurezza.Avuoto  THEN
			QuotaFuoriIngombro_Z_AVUOTO_CCENTRALE := AltezzaDiIngombroArea_CCENTRALE + TCPParameter.Z + OffsetSicurezza.Avuoto;
		END_IF
	END_FOR			
		(* Valuto I Pick-Point *)
		(*FOR P:=1 TO MAXPICKPOINT DO
			AltezzaDiIngombroPuntiPrelievo := 0;
			IF  WorkPickPoint^[P].Zh + WorkPickPointState^[P].ZDim >= WorkPickPointDimension[P].Zdim THEN // Se Altezza orrizzontale Ribaltino + Zpacco >= Ingombro Verticale Ribaltino
				AltezzaDiIngombroPuntiPrelievo := WorkPickPoint^[P].Zh + WorkPickPointState^[P].ZDim;
			END_IF
			IF WorkPickPoint^[P].Zv + WorkPickPointState^[P].ZTilter + WorkPickPointState^[P].YDim >= WorkPickPointDimension[P].Zdim THEN // Se Altezza Vertivale Ribaltino + Quota Fermo + Ypacco >= Ingombro Verticale Ribaltino
				AltezzaDiIngombroPuntiPrelievo := WorkPickPoint^[P].Zv + WorkPickPointState^[P].ZTilter + WorkPickPointState^[P].YDim;
			END_IF
			IF WorkPickPointDimension[P].Zdim >= AltezzaDiIngombroPuntiPrelievo THEN //Se Ingombro Verticale Ribaltino >= Dell'ingombro valutato sopra
				AltezzaDiIngombroPuntiPrelievo := WorkPickPointDimension[P].Zdim;
			END_IF
			IF WAPARTENZA = NPOSTAZIONE_PRIMADELPUNTODIPREL THEN //Se sono nella posizione 7 valuto l'altezza del ribaltino "REALE", con o senza pacco
				IF QuotaAnticipoDinamicaZ_VersoRiposo <= AltezzaDiIngombroPuntiPrelievo + TCPParameter.Z + OffsetSicurezza.Avuoto THEN //Se Quota fuori ingombro <= dell' ingombro del punto di prelievo
					QuotaAnticipoDinamicaZ_VersoRiposo := AltezzaDiIngombroPuntiPrelievo + TCPParameter.Z + OffsetSicurezza.Avuoto;
				END_IF
			ELSE		//Se non sono nella WA 7, do una quota fittizzia, inferiore all'altezza del ribaltino "reale"
				IF QuotaAnticipoDinamicaZ_VersoRiposo <= AltezzaDiIngombroPuntiPrelievo + TCPParameter.Z + OffsetSicurezzaAnticipoMovimenti.OffsetSicurezzaAnticipo_Z - 300 THEN
					QuotaAnticipoDinamicaZ_VersoRiposo := AltezzaDiIngombroPuntiPrelievo + WorkPickPointState^[P].YDim + TCPParameter.Z + OffsetSicurezzaAnticipoMovimenti.OffsetSicurezzaAnticipo_Z - 300;
				END_IF
			END_IF
		END_FOR*)
	//END_IF
	IF ModuleAX_Z^.Ax^.Status.ActPosition >= QuotaAnticipoDinamicaZ_VersoRiposo THEN
		QuotaAnticipoDinamicaZ_Raggiunta := TRUE;
	ELSE
		QuotaAnticipoDinamicaZ_Raggiunta := FALSE;
	END_IF



END_IF*)
END_ACTION

ACTION CalcolaIngombroWALungoX_Pal:
								
AltezzaDiIngombroArea_CCENTRALE := 0;
AltezzaDiIngombroArea_CESTERNO := 0;
AltezzaDiIngombroArea_CESTERNO := 0;
FOR wa := 1 TO MAXAREAPRESENT DO
	
	CASE WorkArea^[wa].Typology OF
		TYPOLOGY_PALLET:
			CASE WorkAreaState^[wa].Supporto.Tipologia OF
					
				PALLET_STANDARD:

					AltezzaDiIngombroArea_CCENTRALE := MAX(AltezzaDiIngombroArea_CCENTRALE, 
															WorkArea^[wa].Z +  MAX(//WorkArea^[wa].Z,
															WorkAreaState^[wa].H,
															WorkAreaState^[wa].HPL,
															WorkAreaState^[wa].Supporto.HMAX,
															WorkAreaState^[wa].Supporto.ZDim));

					AltezzaDiIngombroArea_CESTERNO	:= AltezzaDiIngombroArea_CCENTRALE;
					AltezzaDiIngombroArea_CINTERNO	:= AltezzaDiIngombroArea_CCENTRALE;
					
				PALLET_ACCOPPIATI:

					AltezzaDiIngombroArea_CCENTRALE := MAX(AltezzaDiIngombroArea_CCENTRALE, 
															WorkArea^[wa].Z +  MAX(//WorkArea^[wa].Z,
															WorkAreaState^[wa].H,
															WorkAreaState^[wa].HPL,
															WorkAreaState^[wa].Supporto.HMAX,
															WorkAreaState^[wa].Supporto.ZDim));

					AltezzaDiIngombroArea_CESTERNO	:= AltezzaDiIngombroArea_CCENTRALE;
					AltezzaDiIngombroArea_CINTERNO	:= AltezzaDiIngombroArea_CCENTRALE;
					
					
				CASSA_STANDARD:
									
					AltezzaDiIngombroArea_CCENTRALE := MAX(AltezzaDiIngombroArea_CCENTRALE, 
															WorkArea^[wa].Z +  MAX(//WorkArea^[wa].Z,
															WorkAreaState^[wa].H,
															WorkAreaState^[wa].HPL,
															WorkAreaState^[wa].Supporto.HMAX,
															WorkAreaState^[wa].Supporto.ZDim));

					AltezzaDiIngombroArea_CESTERNO	:= AltezzaDiIngombroArea_CCENTRALE;
					AltezzaDiIngombroArea_CINTERNO	:= AltezzaDiIngombroArea_CCENTRALE;
					
					
				CAVALLETTO:
					AltezzaDiIngombroArea_CCENTRALE := MAX(AltezzaDiIngombroArea_CCENTRALE, 
															WorkArea^[wa].Z,
															//WorkAreaState^[wa].Supporto.HMAX,
															WorkAreaState^[wa].Supporto.ZDim);

					AltezzaDiIngombroArea_CESTERNO	:= MAX(AltezzaDiIngombroArea_CESTERNO,
															WorkArea^[wa].Z,
															//WorkAreaState^[wa].WorkPickPointTransportState.Supporto.HMAX,
															WorkAreaState^[wa].Supporto.ZDim);

					AltezzaDiIngombroArea_CINTERNO	:= AltezzaDiIngombroArea_CESTERNO;
					
				BUNDLE:
					AltezzaDiIngombroArea_CCENTRALE := MAX(AltezzaDiIngombroArea_CCENTRALE, 
															WorkArea^[wa].Z,
															//WorkAreaState^[wa].Supporto.HMAX,
															WorkAreaState^[wa].Supporto.ZDim);

					AltezzaDiIngombroArea_CESTERNO	:= MAX(AltezzaDiIngombroArea_CESTERNO,
															WorkArea^[wa].Z,
															//WorkAreaState^[wa].WorkPickPointTransportState.Supporto.HMAX,
															WorkAreaState^[wa].Supporto.ZDim);

					AltezzaDiIngombroArea_CINTERNO	:= AltezzaDiIngombroArea_CESTERNO;
						
				ELSE
					AltezzaDiIngombroArea_CCENTRALE := WorkArea^[wa].Z;//Fisso l'altezza ad una quota di default
			END_CASE
						
		TYPOLOGY_LAYER:
			AltezzaDiIngombroArea_CCENTRALE := MAX(AltezzaDiIngombroArea_CCENTRALE,
													WorkArea^[wa].Z,
													WorkAreaState^[wa].H,
													WorkAreaState^[wa].HPL);

			AltezzaDiIngombroArea_CESTERNO	:= AltezzaDiIngombroArea_CCENTRALE;
			AltezzaDiIngombroArea_CINTERNO	:= AltezzaDiIngombroArea_CCENTRALE;
		
		TYPOLOGY_EXTERNAL_DEPPREL:
			AltezzaDiIngombroArea_CCENTRALE := AltezzaDiIngombroArea_CCENTRALE;
					
		TYPOLOGY_OVER_TRANSPORT:
			CASE WorkAreaState^[wa].Supporto.Tipologia OF
					
				PALLET_STANDARD:

					AltezzaDiIngombroArea_CCENTRALE := MAX(AltezzaDiIngombroArea_CCENTRALE, 
															WorkArea^[wa].Z +  MAX(//WorkArea^[wa].Z,
															WorkAreaState^[wa].H,
															WorkAreaState^[wa].HPL,
															WorkAreaState^[wa].Supporto.HMAX,
															WorkAreaState^[wa].Supporto.ZDim));

					AltezzaDiIngombroArea_CESTERNO	:= AltezzaDiIngombroArea_CCENTRALE;
					AltezzaDiIngombroArea_CINTERNO	:= AltezzaDiIngombroArea_CCENTRALE;
					
				PALLET_ACCOPPIATI:

					AltezzaDiIngombroArea_CCENTRALE := MAX(AltezzaDiIngombroArea_CCENTRALE, 
															WorkArea^[wa].Z +  MAX(//WorkArea^[wa].Z,
															WorkAreaState^[wa].H,
															WorkAreaState^[wa].HPL,
															WorkAreaState^[wa].Supporto.HMAX,
															WorkAreaState^[wa].Supporto.ZDim));

					AltezzaDiIngombroArea_CESTERNO	:= AltezzaDiIngombroArea_CCENTRALE;
					AltezzaDiIngombroArea_CINTERNO	:= AltezzaDiIngombroArea_CCENTRALE;
	
				CASSA_STANDARD:
									
					AltezzaDiIngombroArea_CCENTRALE := MAX(AltezzaDiIngombroArea_CCENTRALE, 
															WorkArea^[wa].Z +  MAX(//WorkArea^[wa].Z,
															WorkAreaState^[wa].H,
															WorkAreaState^[wa].HPL,
															WorkAreaState^[wa].Supporto.HMAX,
															WorkAreaState^[wa].Supporto.ZDim));

					AltezzaDiIngombroArea_CESTERNO	:= AltezzaDiIngombroArea_CCENTRALE;
					AltezzaDiIngombroArea_CINTERNO	:= AltezzaDiIngombroArea_CCENTRALE;
					
					
				CAVALLETTO:
					AltezzaDiIngombroArea_CCENTRALE := MAX(AltezzaDiIngombroArea_CCENTRALE, 
															WorkArea^[wa].Z,
															WorkAreaState^[wa].Supporto.HMAX,
															WorkAreaState^[wa].Supporto.ZDim);

					AltezzaDiIngombroArea_CESTERNO	:= MAX(AltezzaDiIngombroArea_CESTERNO,
															WorkArea^[wa].Z,
															//WorkAreaState^[wa].WorkPickPointTransportState.Supporto.HMAX,
															WorkAreaState^[wa].Supporto.ZDim);

					AltezzaDiIngombroArea_CINTERNO	:= AltezzaDiIngombroArea_CESTERNO;
					
				BUNDLE:
					AltezzaDiIngombroArea_CCENTRALE := MAX(AltezzaDiIngombroArea_CCENTRALE, 
															WorkArea^[wa].Z,
															WorkAreaState^[wa].Supporto.HMAX,
															WorkAreaState^[wa].Supporto.ZDim);

					AltezzaDiIngombroArea_CESTERNO	:= MAX(AltezzaDiIngombroArea_CESTERNO,
															WorkArea^[wa].Z,
															//WorkAreaState^[wa].WorkPickPointTransportState.Supporto.HMAX,
															WorkAreaState^[wa].Supporto.ZDim);

					AltezzaDiIngombroArea_CINTERNO	:= AltezzaDiIngombroArea_CESTERNO;
				
				ELSE
					AltezzaDiIngombroArea_CCENTRALE := WorkArea^[wa].Z;//Fisso l'altezza ad una quota di default
			END_CASE
	END_CASE															
END_FOR
END_ACTION

ACTION CalcolaIngombroWALungoY:
AltezzaDiIngombroArea_CCENTRALE := 0;
AltezzaDiIngombroArea_CESTERNO := 0;
AltezzaDiIngombroArea_CESTERNO := 0;
FOR wa := 1 TO MAXAREAPRESENT DO
	IF AbilitaValutazioneFISuSingolaWA AND NumeroWAValutazioneFISingolaPostazione > 0 THEN
		wa := NumeroWAValutazioneFISingolaPostazione; 	
	END_IF
	CASE WorkArea^[wa].Typology OF
		TYPOLOGY_PALLET:
			CASE WorkAreaState^[wa].TransportState.Supporto.Tipologia OF
					
				PALLET_STANDARD:

					AltezzaDiIngombroArea_CCENTRALE := MAX(AltezzaDiIngombroArea_CCENTRALE, 
															WorkArea^[wa].Z +  MAX(//WorkArea^[wa].Z,
															WorkAreaState^[wa].H,
															WorkAreaState^[wa].HPL,
															WorkAreaState^[wa].TransportState.Supporto.HMAX,
															WorkAreaState^[wa].TransportState.Supporto.ZDim));

					AltezzaDiIngombroArea_CESTERNO	:= AltezzaDiIngombroArea_CCENTRALE;
					AltezzaDiIngombroArea_CINTERNO	:= AltezzaDiIngombroArea_CCENTRALE;
				
				PALLET_ACCOPPIATI:

					AltezzaDiIngombroArea_CCENTRALE := MAX(AltezzaDiIngombroArea_CCENTRALE, 
															WorkArea^[wa].Z +  MAX(//WorkArea^[wa].Z,
															WorkAreaState^[wa].H,
															WorkAreaState^[wa].HPL,
															WorkAreaState^[wa].TransportState.Supporto.HMAX,
															WorkAreaState^[wa].TransportState.Supporto.ZDim));

					AltezzaDiIngombroArea_CESTERNO	:= AltezzaDiIngombroArea_CCENTRALE;
					AltezzaDiIngombroArea_CINTERNO	:= AltezzaDiIngombroArea_CCENTRALE;				
	
				CASSA_STANDARD:
									
					AltezzaDiIngombroArea_CCENTRALE := MAX(AltezzaDiIngombroArea_CCENTRALE, 
															WorkArea^[wa].Z +  MAX(//WorkArea^[wa].Z,
															WorkAreaState^[wa].H,
															WorkAreaState^[wa].HPL,
															WorkAreaState^[wa].TransportState.Supporto.HMAX,
															WorkAreaState^[wa].TransportState.Supporto.ZDim));

					AltezzaDiIngombroArea_CESTERNO	:= AltezzaDiIngombroArea_CCENTRALE;
					AltezzaDiIngombroArea_CINTERNO	:= AltezzaDiIngombroArea_CCENTRALE;
					
					
				CAVALLETTO:
					AltezzaDiIngombroArea_CCENTRALE := MAX(AltezzaDiIngombroArea_CCENTRALE, 
															WorkArea^[wa].Z,
															//WorkAreaState^[wa].WorkPickPointTransportState.Supporto.HMAX,
															WorkAreaState^[wa].TransportState.Supporto.ZDim);

					AltezzaDiIngombroArea_CESTERNO	:= MAX(AltezzaDiIngombroArea_CESTERNO,
															WorkArea^[wa].Z,
															//WorkAreaState^[wa].WorkPickPointTransportState.Supporto.HMAX,
															WorkAreaState^[wa].TransportState.Supporto.ZDim);

					AltezzaDiIngombroArea_CINTERNO	:= AltezzaDiIngombroArea_CESTERNO;
				
				BUNDLE:
					AltezzaDiIngombroArea_CCENTRALE := MAX(AltezzaDiIngombroArea_CCENTRALE, 
															WorkArea^[wa].Z,
															//WorkAreaState^[wa].WorkPickPointTransportState.Supporto.HMAX,
															WorkAreaState^[wa].TransportState.Supporto.ZDim);

					AltezzaDiIngombroArea_CESTERNO	:= MAX(AltezzaDiIngombroArea_CESTERNO,
															WorkArea^[wa].Z,
															//WorkAreaState^[wa].WorkPickPointTransportState.Supporto.HMAX,
															WorkAreaState^[wa].TransportState.Supporto.ZDim);

					AltezzaDiIngombroArea_CINTERNO	:= AltezzaDiIngombroArea_CESTERNO;
					
